ABB RobotStudio station: Task2_DONE_and_DEMOed.rspag

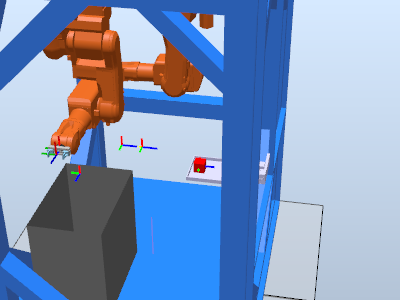
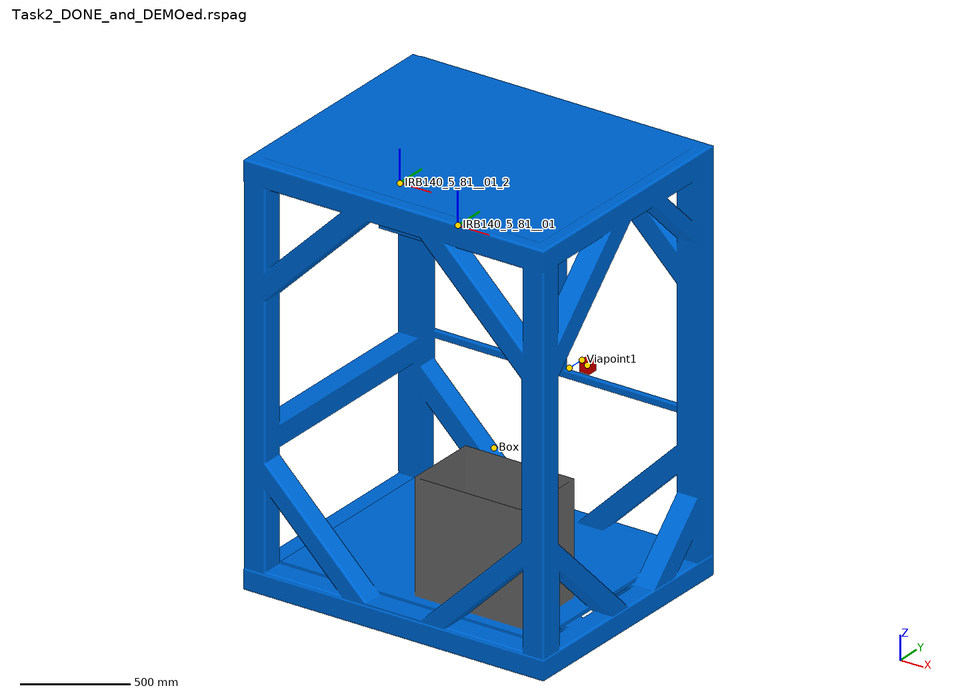
[picture v1: parts stored in the station drawn from their meshes, with robot base, taught points and paths (robot models come from the ABB library and are not in the file)]
--- station ---
Station LCFA_profile (saved by RobotStudio 22.2.10013.1)
Controller ALab_CellC_v1.0_4, task T_ROB2: task frame (RAPID world) sits at (78, -270, 2017) mm, rotated rx 180 ry 0 rz 0 deg in the station
Controller ALab_CellC_v1.0_4, task T_ROB1: task frame (RAPID world) sits at (78, -270, 2017) mm, rotated rx 180 ry 0 rz 0 deg in the station
Controller ALab_CellC_v1.0_4
  mechanical unit ROB_1: IRB140_5_81__01, 6 joints, base frame (0, 0, 0) mm
  mechanical unit ROB_2: IRB140_5_81__01_2, 6 joints, base frame (-596.17, -392.32, 108.97) mm, rotated rx -0.04 ry -0.66 rz 87.49 deg
Layout (positions relative to the parent item):
  - robotcage [part] at (0, 0, 87) mm, size 1670.4 x 1374.8 x 2180.4 mm
  - SampleTray [mechanism, from Libraries\SampleTray.rslib] at (263, 650, 160) mm; joint values [0] (rad or m)
  - IRB140_5_81__01 [mechanism, from Robots\IRB140_5_81__01.rslib] at (78, -270, 2017) mm, rotated rx 180 ry 0 rz 0 deg; joint values [0, 0, 0, 0, 0, 0] (rad or m)
  - IRB140_5_81__01_2 [mechanism, from Robots\IRB140_5_81__01.rslib] at (-518.17, 122.32, 1908.03) mm, rotated rx 179.96 ry 0.66 rz -87.49 deg; joint values [0, 0, 0, 0, 0, 0] (rad or m)
  - Gripper [mechanism, from Libraries\Gripper.rslib] at (593, -270, 1305) mm, rotated rx 0 ry -90 rz -180 deg; joint values [0] (rad or m)
  - Rubic Cube [part] at (76, 83.24, 1430.78) mm, rotated rx 180 ry 0 rz 90 deg, size 55 x 55 x 55 mm
  - Rubic Cube Simulation  [smart component]
      signals: DI DI_Open, DI DI_Close
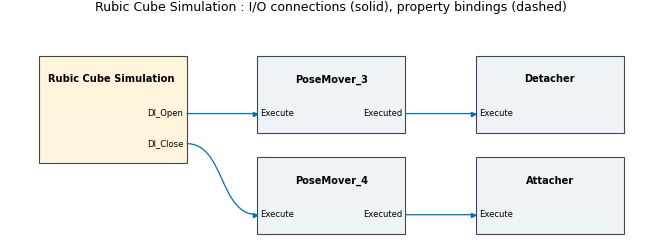
      connections:
        Rubic Cube Simulation .DI_Open -> PoseMover_3.Execute
        Rubic Cube Simulation .DI_Close -> PoseMover_4.Execute
        PoseMover_4.Executed -> Attacher.Execute
        PoseMover_3.Executed -> Detacher.Execute
    - PoseMover_3 [smart component, from Components\PoseMover.rslib]
        properties: Mechanism=Gripper; Pose=1; Duration=1
    - PoseMover_4 [smart component, from Components\PoseMover.rslib]
        properties: Mechanism=Gripper; Pose=2; Duration=1
    - Attacher [smart component, from Components\Attacher.rslib]
        properties: Parent=Gripper; Flange=0; Child=Rubic Cube; Mount=false; Offset=[0 0 0]; Orientation=[0 0 0]
    - Detacher [smart component, from Components\Detacher.rslib]
        properties: Child=Rubic Cube; KeepPosition=false
  - Box_1 [part] at (0, -500, 220) mm, size 600 x 400 x 0 mm
  - Box_2 [part] at (0, -500, 220) mm, rotated rx 90 ry 0 rz 0 deg, size 600 x 600 x 400 mm
  - Box_3 [part] at (0, -500, 820) mm, rotated rx 0 ry 90 rz 0 deg, size 600 x 400 x 600 mm
Attachment: Gripper is attached to IRB140_5_81__01 / Link6
EventTableEntry 4073: Group=, Trigger=AND 4074, Actions=[pose1 4075], Comment=, ActivationMode=2, Cyclic=false
EventTableTriggerLogic 4074: layoutX=167, layoutY=76, Operand1=AND 4076, Operand2=AND 4081, Operator=0, Delay=1000
EventTableActionIO 4075: IOValue=[-1], IRC5Controller=? -1, SignalTarget=LCFA_profile 1
EventTableTriggerLogic 4076: layoutX=94, layoutY=38, Operand1=cellC_gripper_horizontal_move 7096, Operand2=cellC_gripper_vertical_move 7097, Operator=0, Delay=1000
EventTableTriggerLogic 4081: layoutX=94, layoutY=109, Operand1=NOT 4082, Operand2=NOT 4084, Operator=0, Delay=1000
EventTableTriggerLogic 4082: layoutX=14, layoutY=96, Operand1=cellC_slider_horizontal_move 6338, Operand2=? -1, Operator=2, Delay=1000
EventTableTriggerLogic 4084: layoutX=9, layoutY=134, Operand1=cellC_slider_vertical_move 6339, Operand2=? -1, Operator=2, Delay=1000
EventTableEntry 4086: Group=, Trigger=AND 4087, Actions=[pose4 4097], Comment=, ActivationMode=2, Cyclic=false
EventTableTriggerLogic 4087: layoutX=194, layoutY=70, Operand1=AND 4088, Operand2=AND 4093, Operator=0, Delay=1000
EventTableTriggerLogic 4088: layoutX=73, layoutY=39, Operand1=cellC_gripper_horizontal_move 7098, Operand2=cellC_gripper_vertical_move 7099, Operator=0, Delay=1000
EventTableTriggerLogic 4093: layoutX=125, layoutY=101, Operand1=NOT 4094, Operand2=cellC_slider_vertical_move 6343, Operator=0, Delay=1000
EventTableTriggerLogic 4094: layoutX=19, layoutY=95, Operand1=cellC_slider_horizontal_move 6342, Operand2=? -1, Operator=2, Delay=1000
EventTableActionIO 4097: IOValue=[-1], IRC5Controller=? -1, SignalTarget=LCFA_profile 1
EventTableEntry 4098: Group=, Trigger=AND 4099, Actions=[pose8 4109], Comment=, ActivationMode=2, Cyclic=false
EventTableTriggerLogic 4099: layoutX=181, layoutY=88, Operand1=AND 4100, Operand2=AND 4105, Operator=0, Delay=1000
EventTableTriggerLogic 4100: layoutX=94, layoutY=47, Operand1=cellC_gripper_horizontal_move 7100, Operand2=cellC_gripper_vertical_move 7101, Operator=0, Delay=1000
EventTableTriggerLogic 4105: layoutX=92, layoutY=128, Operand1=cellC_slider_horizontal_move 6347, Operand2=NOT 4107, Operator=0, Delay=1000
EventTableTriggerLogic 4107: layoutX=18, layoutY=134, Operand1=cellC_slider_vertical_move 6346, Operand2=? -1, Operator=2, Delay=1000
EventTableActionIO 4109: IOValue=[-1], IRC5Controller=? -1, SignalTarget=LCFA_profile 1
EventTableEntry 4110: Group=, Trigger=AND 4111, Actions=[pose11 4120], Comment=, ActivationMode=2, Cyclic=false
EventTableTriggerLogic 4111: layoutX=165, layoutY=70, Operand1=AND 4112, Operand2=AND 4117, Operator=0, Delay=1000
EventTableTriggerLogic 4112: layoutX=93, layoutY=33, Operand1=cellC_gripper_horizontal_move 7102, Operand2=cellC_gripper_vertical_move 7103, Operator=0, Delay=1000
EventTableTriggerLogic 4117: layoutX=93, layoutY=131, Operand1=cellC_slider_horizontal_move 6350, Operand2=cellC_slider_vertical_move 6351, Operator=0, Delay=1000
EventTableActionIO 4120: IOValue=[-1], IRC5Controller=? -1, SignalTarget=LCFA_profile 1
EventTableEntry 4121: Group=, Trigger=AND 4122, Actions=[pose17 4132], Comment=, ActivationMode=2, Cyclic=false
EventTableTriggerLogic 4122: layoutX=217, layoutY=77, Operand1=AND 4123, Operand2=AND 4127, Operator=0, Delay=1000
EventTableTriggerLogic 4123: layoutX=119, layoutY=36, Operand1=cellC_gripper_horizontal_move 7960, Operand2=NOT 7105, Operator=0, Delay=1000
EventTableTriggerLogic 4127: layoutX=112, layoutY=96, Operand1=NOT 4128, Operand2=NOT 4130, Operator=0, Delay=1000
EventTableTriggerLogic 4128: layoutX=40, layoutY=96, Operand1=cellC_slider_horizontal_move 7961, Operand2=? -1, Operator=2, Delay=1000
EventTableTriggerLogic 4130: layoutX=35, layoutY=134, Operand1=cellC_slider_vertical_move 7962, Operand2=? -1, Operator=2, Delay=1000
EventTableActionIO 4132: IOValue=[-1], IRC5Controller=? -1, SignalTarget=LCFA_profile 1
EventTableEntry 4133: Group=, Trigger=AND 4134, Actions=[pose16 4143], Comment=, ActivationMode=2, Cyclic=false
EventTableTriggerLogic 4134: layoutX=168, layoutY=84, Operand1=AND 4135, Operand2=AND 4139, Operator=0, Delay=1000
EventTableTriggerLogic 4135: layoutX=90, layoutY=31, Operand1=cellC_gripper_horizontal_move 7106, Operand2=NOT 7107, Operator=0, Delay=1000
EventTableTriggerLogic 4139: layoutX=77, layoutY=109, Operand1=NOT 4253, Operand2=cellC_slider_vertical_move 6671, Operator=0, Delay=1000
EventTableActionIO 4143: IOValue=[-1], IRC5Controller=? -1, SignalTarget=LCFA_profile 1
EventTableEntry 4144: Group=, Trigger=AND 4145, Actions=[pose10 4154], Comment=, ActivationMode=2, Cyclic=false
EventTableTriggerLogic 4145: layoutX=219, layoutY=73, Operand1=AND 4146, Operand2=AND 4150, Operator=0, Delay=1000
EventTableTriggerLogic 4146: layoutX=143, layoutY=36, Operand1=cellC_gripper_horizontal_move 7964, Operand2=NOT 7110, Operator=0, Delay=1000
EventTableTriggerLogic 4150: layoutX=143, layoutY=107, Operand1=cellC_slider_horizontal_move 7966, Operand2=NOT 4152, Operator=0, Delay=1000
EventTableTriggerLogic 4152: layoutX=16, layoutY=136, Operand1=cellC_slider_vertical_move 7965, Operand2=? -1, Operator=2, Delay=1000
EventTableActionIO 4154: IOValue=[-1], IRC5Controller=? -1, SignalTarget=LCFA_profile 1
EventTableEntry 4155: Group=, Trigger=AND 4156, Actions=[pose14 4164], Comment=, ActivationMode=2, Cyclic=false
EventTableTriggerLogic 4156: layoutX=203, layoutY=67, Operand1=AND 4157, Operand2=AND 4161, Operator=0, Delay=1000
EventTableTriggerLogic 4157: layoutX=135, layoutY=41, Operand1=cellC_gripper_horizontal_move 7968, Operand2=NOT 7112, Operator=0, Delay=1000
EventTableTriggerLogic 4161: layoutX=132, layoutY=113, Operand1=cellC_slider_horizontal_move 7969, Operand2=cellC_slider_vertical_move 7970, Operator=0, Delay=1000
EventTableActionIO 4164: IOValue=[-1], IRC5Controller=? -1, SignalTarget=LCFA_profile 1
EventTableEntry 4165: Group=, Trigger=AND 4166, Actions=[pose2 4176], Comment=, ActivationMode=2, Cyclic=false
EventTableTriggerLogic 4166: layoutX=220, layoutY=69, Operand1=AND 4167, Operand2=AND 4171, Operator=0, Delay=1000
EventTableTriggerLogic 4167: layoutX=125, layoutY=14, Operand1=NOT 8003, Operand2=cellC_gripper_vertical_move 7972, Operator=0, Delay=1000
EventTableTriggerLogic 4171: layoutX=124, layoutY=95, Operand1=NOT 4172, Operand2=NOT 4174, Operator=0, Delay=1000
EventTableTriggerLogic 4172: layoutX=13, layoutY=97, Operand1=cellC_slider_horizontal_move 7973, Operand2=? -1, Operator=2, Delay=1000
EventTableTriggerLogic 4174: layoutX=11, layoutY=134, Operand1=cellC_slider_vertical_move 7974, Operand2=? -1, Operator=2, Delay=1000
EventTableActionIO 4176: IOValue=[-1], IRC5Controller=? -1, SignalTarget=LCFA_profile 1
EventTableEntry 4177: Group=, Trigger=AND 4178, Actions=[pose5 4187], Comment=, ActivationMode=2, Cyclic=false
EventTableTriggerLogic 4178: layoutX=243, layoutY=55, Operand1=AND 4179, Operand2=AND 4183, Operator=0, Delay=1000
EventTableTriggerLogic 4179: layoutX=162, layoutY=28, Operand1=NOT 8005, Operand2=cellC_gripper_vertical_move 7976, Operator=0, Delay=1000
EventTableTriggerLogic 4183: layoutX=173, layoutY=138, Operand1=NOT 4184, Operand2=cellC_slider_vertical_move 7978, Operator=0, Delay=1000
EventTableTriggerLogic 4184: layoutX=18, layoutY=95, Operand1=cellC_slider_horizontal_move 7977, Operand2=? -1, Operator=2, Delay=1000
EventTableActionIO 4187: IOValue=[-1], IRC5Controller=? -1, SignalTarget=LCFA_profile 1
EventTableEntry 4188: Group=, Trigger=AND 4189, Actions=[pose9 4198], Comment=, ActivationMode=2, Cyclic=false
EventTableTriggerLogic 4189: layoutX=204, layoutY=112, Operand1=AND 4190, Operand2=AND 4194, Operator=0, Delay=1000
EventTableTriggerLogic 4190: layoutX=108, layoutY=30, Operand1=NOT 8007, Operand2=cellC_gripper_vertical_move 7980, Operator=0, Delay=1000
EventTableTriggerLogic 4194: layoutX=108, layoutY=141, Operand1=cellC_slider_horizontal_move 7982, Operand2=NOT 4196, Operator=0, Delay=1000
EventTableTriggerLogic 4196: layoutX=26, layoutY=161, Operand1=cellC_slider_vertical_move 7981, Operand2=? -1, Operator=2, Delay=1000
EventTableActionIO 4198: IOValue=[-1], IRC5Controller=? -1, SignalTarget=LCFA_profile 1
EventTableEntry 4199: Group=, Trigger=AND 4200, Actions=[pose12 4208], Comment=, ActivationMode=2, Cyclic=false
EventTableTriggerLogic 4200: layoutX=245, layoutY=97, Operand1=AND 4201, Operand2=AND 4205, Operator=0, Delay=1000
EventTableTriggerLogic 4201: layoutX=182, layoutY=72, Operand1=NOT 8009, Operand2=cellC_gripper_vertical_move 7984, Operator=0, Delay=1000
EventTableTriggerLogic 4205: layoutX=189, layoutY=131, Operand1=cellC_slider_horizontal_move 7985, Operand2=cellC_slider_vertical_move 7986, Operator=0, Delay=1000
EventTableActionIO 4208: IOValue=[-1], IRC5Controller=? -1, SignalTarget=LCFA_profile 1
EventTableEntry 4209: Group=, Trigger=AND 4210, Actions=[pose3 4219], Comment=, ActivationMode=2, Cyclic=false
EventTableTriggerLogic 4210: layoutX=234, layoutY=61, Operand1=AND 4211, Operand2=AND 4214, Operator=0, Delay=1000
EventTableTriggerLogic 4211: layoutX=80, layoutY=23, Operand1=NOT 7117, Operand2=NOT 7118, Operator=0, Delay=1000
EventTableTriggerLogic 4214: layoutX=88, layoutY=113, Operand1=NOT 4215, Operand2=NOT 4217, Operator=0, Delay=1000
EventTableTriggerLogic 4215: layoutX=16, layoutY=85, Operand1=cellC_slider_horizontal_move 7989, Operand2=? -1, Operator=2, Delay=1000
EventTableTriggerLogic 4217: layoutX=33, layoutY=125, Operand1=cellC_slider_vertical_move 7990, Operand2=? -1, Operator=2, Delay=1000
EventTableActionIO 4219: IOValue=[-1], IRC5Controller=? -1, SignalTarget=LCFA_profile 1
EventTableEntry 4220: Group=, Trigger=AND 4221, Actions=[pose6 4229], Comment=, ActivationMode=2, Cyclic=false
EventTableTriggerLogic 4221: layoutX=192, layoutY=87, Operand1=AND 4222, Operand2=AND 4225, Operator=0, Delay=1000
EventTableTriggerLogic 4222: layoutX=118, layoutY=38, Operand1=NOT 7119, Operand2=NOT 7120, Operator=0, Delay=1000
EventTableTriggerLogic 4225: layoutX=113, layoutY=118, Operand1=NOT 4226, Operand2=cellC_slider_vertical_move 7994, Operator=0, Delay=1000
EventTableTriggerLogic 4226: layoutX=14, layoutY=101, Operand1=cellC_slider_horizontal_move 7993, Operand2=? -1, Operator=2, Delay=1000
EventTableActionIO 4229: IOValue=[-1], IRC5Controller=? -1, SignalTarget=LCFA_profile 1
EventTableEntry 4230: Group=, Trigger=AND 4231, Actions=[pose7 4239], Comment=, ActivationMode=2, Cyclic=false
EventTableTriggerLogic 4231: layoutX=212, layoutY=64, Operand1=AND 4232, Operand2=AND 4235, Operator=0, Delay=1000
EventTableTriggerLogic 4232: layoutX=113, layoutY=37, Operand1=NOT 7121, Operand2=NOT 7122, Operator=0, Delay=1000
EventTableTriggerLogic 4235: layoutX=113, layoutY=104, Operand1=cellC_slider_horizontal_move 7998, Operand2=NOT 4237, Operator=0, Delay=1000
EventTableTriggerLogic 4237: layoutX=13, layoutY=128, Operand1=cellC_slider_vertical_move 7997, Operand2=? -1, Operator=2, Delay=1000
EventTableActionIO 4239: IOValue=[-1], IRC5Controller=? -1, SignalTarget=LCFA_profile 1
EventTableEntry 4240: Group=, Trigger=AND 4241, Actions=[pose13 4248], Comment=, ActivationMode=2, Cyclic=false
EventTableTriggerLogic 4241: layoutX=160, layoutY=73, Operand1=AND 4242, Operand2=AND 4245, Operator=0, Delay=1000
EventTableTriggerLogic 4242: layoutX=68, layoutY=38, Operand1=NOT 7123, Operand2=NOT 7124, Operator=0, Delay=1000
EventTableTriggerLogic 4245: layoutX=67, layoutY=107, Operand1=cellC_slider_horizontal_move 8001, Operand2=cellC_slider_vertical_move 8002, Operator=0, Delay=1000
EventTableActionIO 4248: IOValue=[-1], IRC5Controller=? -1, SignalTarget=LCFA_profile 1
EventTableTriggerLogic 4253: layoutX=22, layoutY=89, Operand1=cellC_slider_horizontal_move 6670, Operand2=? -1, Operator=2, Delay=1000
EventTableEntry 4262: Group=, Trigger=AND 4263, Actions=[conv1_buffer6 4271], Comment=, ActivationMode=2, Cyclic=false
EventTableTriggerLogic 4263: layoutX=153, layoutY=73, Operand1=AND 4264, Operand2=NOT 4269, Operator=0, Delay=1000
EventTableTriggerLogic 4264: layoutX=80, layoutY=34, Operand1=NOT 4265, Operand2=NOT 4267, Operator=0, Delay=1000
EventTableTriggerLogic 4265: layoutX=8, layoutY=16, Operand1=conv1_buffer_horizontal_open 6327, Operand2=? -1, Operator=2, Delay=1000
EventTableTriggerLogic 4267: layoutX=9, layoutY=52, Operand1=conv1_buffer_lower_go_up 6328, Operand2=? -1, Operator=2, Delay=1000
EventTableTriggerLogic 4269: layoutX=9, layoutY=86, Operand1=conv1_buffer_upper_go_down 6329, Operand2=? -1, Operator=2, Delay=1000
EventTableActionIO 4271: IOValue=[-1], IRC5Controller=? -1, SignalTarget=LCFA_profile 1
EventTableEntry 4272: Group=, Trigger=AND 4273, Actions=[conv1_buffer5 4280], Comment=, ActivationMode=2, Cyclic=false
EventTableTriggerLogic 4273: layoutX=133, layoutY=81, Operand1=AND 4274, Operand2=conv1_buffer_upper_go_down 6332, Operator=0, Delay=1000
EventTableTriggerLogic 4274: layoutX=93, layoutY=26, Operand1=NOT 4275, Operand2=NOT 4277, Operator=0, Delay=1000
EventTableTriggerLogic 4275: layoutX=8, layoutY=16, Operand1=conv1_buffer_horizontal_open 6330, Operand2=? -1, Operator=2, Delay=1000
EventTableTriggerLogic 4277: layoutX=9, layoutY=53, Operand1=conv1_buffer_lower_go_up 6331, Operand2=? -1, Operator=2, Delay=1000
EventTableActionIO 4280: IOValue=[-1], IRC5Controller=? -1, SignalTarget=LCFA_profile 1
EventTableEntry 4281: Group=, Trigger=AND 4282, Actions=[conv1_buffer8 4289], Comment=, ActivationMode=2, Cyclic=false
EventTableTriggerLogic 4282: layoutX=184, layoutY=91, Operand1=AND 4283, Operand2=NOT 4287, Operator=0, Delay=1000
EventTableTriggerLogic 4283: layoutX=106, layoutY=52, Operand1=NOT 4284, Operand2=conv1_buffer_lower_go_up 6334, Operator=0, Delay=1000
EventTableTriggerLogic 4284: layoutX=13, layoutY=17, Operand1=conv1_buffer_horizontal_open 6333, Operand2=? -1, Operator=2, Delay=1000
EventTableTriggerLogic 4287: layoutX=23, layoutY=94, Operand1=conv1_buffer_upper_go_down 6335, Operand2=? -1, Operator=2, Delay=1000
EventTableActionIO 4289: IOValue=[-1], IRC5Controller=? -1, SignalTarget=LCFA_profile 1
EventTableEntry 4290: Group=, Trigger=AND 4291, Actions=[conv1_buffer7 4297], Comment=, ActivationMode=2, Cyclic=false
EventTableTriggerLogic 4291: layoutX=211, layoutY=90, Operand1=AND 4292, Operand2=conv1_buffer_upper_go_down 6282, Operator=0, Delay=1000
EventTableTriggerLogic 4292: layoutX=106, layoutY=24, Operand1=NOT 4293, Operand2=conv1_buffer_lower_go_up 6281, Operator=0, Delay=1000
EventTableTriggerLogic 4293: layoutX=35, layoutY=17, Operand1=conv1_buffer_horizontal_open 6280, Operand2=? -1, Operator=2, Delay=1000
EventTableActionIO 4297: IOValue=[-1], IRC5Controller=? -1, SignalTarget=LCFA_profile 1
EventTableEntry 4298: Group=, Trigger=AND 4299, Actions=[conv1_buffer2 4306], Comment=, ActivationMode=2, Cyclic=false
EventTableTriggerLogic 4299: layoutX=226, layoutY=110, Operand1=AND 4300, Operand2=NOT 4304, Operator=0, Delay=1000
EventTableTriggerLogic 4300: layoutX=93, layoutY=30, Operand1=conv1_buffer_horizontal_open 6284, Operand2=NOT 4302, Operator=0, Delay=1000
EventTableTriggerLogic 4302: layoutX=30, layoutY=56, Operand1=conv1_buffer_lower_go_up 6283, Operand2=? -1, Operator=2, Delay=1000
EventTableTriggerLogic 4304: layoutX=17, layoutY=96, Operand1=conv1_buffer_upper_go_down 6285, Operand2=? -1, Operator=2, Delay=1000
EventTableActionIO 4306: IOValue=[-1], IRC5Controller=? -1, SignalTarget=LCFA_profile 1
EventTableEntry 4307: Group=, Trigger=AND 4308, Actions=[conv1_buffer1 4314], Comment=, ActivationMode=2, Cyclic=false
EventTableTriggerLogic 4308: layoutX=164, layoutY=68, Operand1=AND 4309, Operand2=conv1_buffer_upper_go_down 6288, Operator=0, Delay=1000
EventTableTriggerLogic 4309: layoutX=96, layoutY=16, Operand1=conv1_buffer_horizontal_open 6287, Operand2=NOT 4311, Operator=0, Delay=1000
EventTableTriggerLogic 4311: layoutX=18, layoutY=46, Operand1=conv1_buffer_lower_go_up 6286, Operand2=? -1, Operator=2, Delay=1000
EventTableActionIO 4314: IOValue=[-1], IRC5Controller=? -1, SignalTarget=LCFA_profile 1
EventTableEntry 4315: Group=, Trigger=AND 4316, Actions=[conv1_buffer4 4322], Comment=, ActivationMode=2, Cyclic=false
EventTableTriggerLogic 4316: layoutX=161, layoutY=63, Operand1=AND 4317, Operand2=NOT 4320, Operator=0, Delay=1000
EventTableTriggerLogic 4317: layoutX=52, layoutY=16, Operand1=conv1_buffer_horizontal_open 6289, Operand2=conv1_buffer_lower_go_up 6290, Operator=0, Delay=1000
EventTableTriggerLogic 4320: layoutX=26, layoutY=137, Operand1=conv1_buffer_upper_go_down 6291, Operand2=? -1, Operator=2, Delay=1000
EventTableActionIO 4322: IOValue=[-1], IRC5Controller=? -1, SignalTarget=LCFA_profile 1
EventTableEntry 4323: Group=, Trigger=AND 4324, Actions=[conv1_buffer3 4329], Comment=, ActivationMode=2, Cyclic=false
EventTableTriggerLogic 4324: layoutX=174, layoutY=87, Operand1=AND 4325, Operand2=conv1_buffer_upper_go_down 6294, Operator=0, Delay=1000
EventTableTriggerLogic 4325: layoutX=74, layoutY=31, Operand1=conv1_buffer_horizontal_open 6292, Operand2=conv1_buffer_lower_go_up 6293, Operator=0, Delay=1000
EventTableActionIO 4329: IOValue=[-1], IRC5Controller=? -1, SignalTarget=LCFA_profile 1
EventTableEntry 4330: Group=, Trigger=AND 4331, Actions=[conv2_buffer6 4339], Comment=, ActivationMode=2, Cyclic=false
EventTableTriggerLogic 4331: layoutX=148, layoutY=98, Operand1=AND 4332, Operand2=NOT 4337, Operator=0, Delay=1000
EventTableTriggerLogic 4332: layoutX=101, layoutY=54, Operand1=NOT 4333, Operand2=NOT 4335, Operator=0, Delay=1000
EventTableTriggerLogic 4333: layoutX=31, layoutY=17, Operand1=conv2_buffer_horizontal_move 6295, Operand2=? -1, Operator=2, Delay=1000
EventTableTriggerLogic 4335: layoutX=32, layoutY=53, Operand1=conv2_buffer_lower_vertical_move 6296, Operand2=? -1, Operator=2, Delay=1000
EventTableTriggerLogic 4337: layoutX=31, layoutY=89, Operand1=conv2_buffer_upper_vertical_move 6297, Operand2=? -1, Operator=2, Delay=1000
EventTableActionIO 4339: IOValue=[-1], IRC5Controller=? -1, SignalTarget=LCFA_profile 1
EventTableEntry 4340: Group=, Trigger=AND 4341, Actions=[conv2_buffer5 4348], Comment=, ActivationMode=2, Cyclic=false
EventTableTriggerLogic 4341: layoutX=206, layoutY=74, Operand1=AND 4342, Operand2=conv2_buffer_upper_vertical_move 6300, Operator=0, Delay=1000
EventTableTriggerLogic 4342: layoutX=94, layoutY=37, Operand1=NOT 4343, Operand2=NOT 4345, Operator=0, Delay=1000
EventTableTriggerLogic 4343: layoutX=13, layoutY=14, Operand1=conv2_buffer_horizontal_move 6298, Operand2=? -1, Operator=2, Delay=1000
EventTableTriggerLogic 4345: layoutX=9, layoutY=56, Operand1=conv2_buffer_lower_vertical_move 6299, Operand2=? -1, Operator=2, Delay=1000
EventTableActionIO 4348: IOValue=[-1], IRC5Controller=? -1, SignalTarget=LCFA_profile 1
EventTableEntry 4349: Group=, Trigger=AND 4350, Actions=[conv2_buffer8 4357], Comment=, ActivationMode=2, Cyclic=false
EventTableTriggerLogic 4350: layoutX=195, layoutY=82, Operand1=AND 4351, Operand2=NOT 4355, Operator=0, Delay=1000
EventTableTriggerLogic 4351: layoutX=67, layoutY=49, Operand1=NOT 4352, Operand2=conv2_buffer_lower_vertical_move 6302, Operator=0, Delay=1000
EventTableTriggerLogic 4352: layoutX=20, layoutY=15, Operand1=conv2_buffer_horizontal_move 6301, Operand2=? -1, Operator=2, Delay=1000
EventTableTriggerLogic 4355: layoutX=20, layoutY=92, Operand1=conv2_buffer_upper_vertical_move 6303, Operand2=? -1, Operator=2, Delay=1000
EventTableActionIO 4357: IOValue=[-1], IRC5Controller=? -1, SignalTarget=LCFA_profile 1
EventTableEntry 4358: Group=, Trigger=AND 4359, Actions=[conv2_buffer7 4365], Comment=, ActivationMode=2, Cyclic=false
EventTableTriggerLogic 4359: layoutX=193, layoutY=94, Operand1=AND 4360, Operand2=conv2_buffer_upper_vertical_move 6306, Operator=0, Delay=1000
EventTableTriggerLogic 4360: layoutX=111, layoutY=44, Operand1=NOT 4361, Operand2=conv2_buffer_lower_vertical_move 6305, Operator=0, Delay=1000
EventTableTriggerLogic 4361: layoutX=48, layoutY=16, Operand1=conv2_buffer_horizontal_move 6304, Operand2=? -1, Operator=2, Delay=1000
EventTableActionIO 4365: IOValue=[-1], IRC5Controller=? -1, SignalTarget=LCFA_profile 1
EventTableEntry 4366: Group=, Trigger=AND 4367, Actions=[conv2_buffer2 4374], Comment=, ActivationMode=2, Cyclic=false
EventTableTriggerLogic 4367: layoutX=210, layoutY=27, Operand1=conv2_buffer_horizontal_move 6309, Operand2=AND 4369, Operator=0, Delay=1000
EventTableTriggerLogic 4369: layoutX=163, layoutY=91, Operand1=NOT 4370, Operand2=NOT 4372, Operator=0, Delay=1000
EventTableTriggerLogic 4370: layoutX=21, layoutY=58, Operand1=conv2_buffer_lower_vertical_move 6307, Operand2=? -1, Operator=2, Delay=1000
EventTableTriggerLogic 4372: layoutX=24, layoutY=96, Operand1=conv2_buffer_upper_vertical_move 6308, Operand2=? -1, Operator=2, Delay=1000
EventTableActionIO 4374: IOValue=[-1], IRC5Controller=? -1, SignalTarget=LCFA_profile 1
EventTableEntry 4375: Group=, Trigger=AND 4376, Actions=[conv2_buffer1 4382], Comment=, ActivationMode=2, Cyclic=false
EventTableTriggerLogic 4376: layoutX=233, layoutY=95, Operand1=AND 4377, Operand2=conv2_buffer_upper_vertical_move 6312, Operator=0, Delay=1000
EventTableTriggerLogic 4377: layoutX=160, layoutY=50, Operand1=conv2_buffer_horizontal_move 6311, Operand2=NOT 4379, Operator=0, Delay=1000
EventTableTriggerLogic 4379: layoutX=37, layoutY=56, Operand1=conv2_buffer_lower_vertical_move 6310, Operand2=? -1, Operator=2, Delay=1000
EventTableActionIO 4382: IOValue=[-1], IRC5Controller=? -1, SignalTarget=LCFA_profile 1
EventTableEntry 4383: Group=, Trigger=AND 4384, Actions=[conv2_buffer4 4390], Comment=, ActivationMode=2, Cyclic=false
EventTableTriggerLogic 4384: layoutX=102, layoutY=69, Operand1=AND 4385, Operand2=NOT 4388, Operator=0, Delay=1000
EventTableTriggerLogic 4385: layoutX=32, layoutY=42, Operand1=conv2_buffer_horizontal_move 6313, Operand2=conv2_buffer_lower_vertical_move 6314, Operator=0, Delay=1000
EventTableTriggerLogic 4388: layoutX=24, layoutY=96, Operand1=conv2_buffer_upper_vertical_move 6315, Operand2=? -1, Operator=2, Delay=1000
EventTableActionIO 4390: IOValue=[-1], IRC5Controller=? -1, SignalTarget=LCFA_profile 1
EventTableEntry 4391: Group=, Trigger=AND 4392, Actions=[conv2_buffer3 4397], Comment=, ActivationMode=2, Cyclic=false
EventTableTriggerLogic 4392: layoutX=97, layoutY=92, Operand1=AND 4393, Operand2=conv2_buffer_upper_vertical_move 6318, Operator=0, Delay=1000
EventTableTriggerLogic 4393: layoutX=42, layoutY=52, Operand1=conv2_buffer_horizontal_move 6316, Operand2=conv2_buffer_lower_vertical_move 6317, Operator=0, Delay=1000
EventTableActionIO 4397: IOValue=[-1], IRC5Controller=? -1, SignalTarget=LCFA_profile 1
EventTableEntry 4398: Group=, Trigger=AND 4399, Actions=[palletHolder1 4404], Comment=, ActivationMode=2, Cyclic=false
EventTableTriggerLogic 4399: layoutX=96, layoutY=16, Operand1=cellC_pallet_holder 7125, Operand2=cellC_pallet_stopper 7126, Operator=0, Delay=1000
EventTableActionIO 4404: IOValue=[-1], IRC5Controller=? -1, SignalTarget=LCFA_profile 1
EventTableEntry 4405: Group=, Trigger=AND 4406, Actions=[palletHolder2 4410], Comment=, ActivationMode=2, Cyclic=false
EventTableTriggerLogic 4406: layoutX=142, layoutY=32, Operand1=NOT 7128, Operand2=cellC_pallet_stopper 7127, Operator=0, Delay=1000
EventTableActionIO 4410: IOValue=[-1], IRC5Controller=? -1, SignalTarget=LCFA_profile 1
EventTableEntry 4411: Group=, Trigger=AND 4412, Actions=[palletHolder4 4415], Comment=, ActivationMode=2, Cyclic=false
EventTableTriggerLogic 4412: layoutX=51, layoutY=46, Operand1=NOT 7130, Operand2=NOT 7132, Operator=0, Delay=1000
EventTableActionIO 4415: IOValue=[-1], IRC5Controller=? -1, SignalTarget=LCFA_profile 1
EventTableEntry 4416: Group=, Trigger=AND 4417, Actions=[palletHolder3 4419], Comment=, ActivationMode=2, Cyclic=false
EventTableTriggerLogic 4417: layoutX=107, layoutY=60, Operand1=cellC_pallet_holder 7134, Operand2=NOT 7135, Operator=0, Delay=1000
EventTableActionIO 4419: IOValue=[-1], IRC5Controller=? -1, SignalTarget=LCFA_profile 1
EventTableEntry 4425: Group=, Trigger=TestPlateDrive 4426, Actions=[EventTableActionMechanicalPose 4427], Comment=, ActivationMode=2, Cyclic=false
EventTableTriggerIO 4426: IOValue=[1], IRC5Controller=? -1, Operator=0, SignalSource=ALab_CellC_v1.0_4 5362
EventTableActionMechanicalPose 4427: VirtualSignal=, Mechanism=SampleTray 568, ToPoseName=HomePosition, VirtualSignalValue=[1]
EventTableTriggerIO 6280: IOValue=[-1], IRC5Controller=? -1, Operator=0, SignalSource=ALab_CellC_v1.0_4 5362
EventTableTriggerIO 6281: IOValue=[-1], IRC5Controller=? -1, Operator=0, SignalSource=ALab_CellC_v1.0_4 5362
EventTableTriggerIO 6282: IOValue=[-1], IRC5Controller=? -1, Operator=0, SignalSource=ALab_CellC_v1.0_4 5362
EventTableTriggerIO 6283: IOValue=[-1], IRC5Controller=? -1, Operator=0, SignalSource=ALab_CellC_v1.0_4 5362
EventTableTriggerIO 6284: IOValue=[-1], IRC5Controller=? -1, Operator=0, SignalSource=ALab_CellC_v1.0_4 5362
EventTableTriggerIO 6285: IOValue=[-1], IRC5Controller=? -1, Operator=0, SignalSource=ALab_CellC_v1.0_4 5362
EventTableTriggerIO 6286: IOValue=[-1], IRC5Controller=? -1, Operator=0, SignalSource=ALab_CellC_v1.0_4 5362
EventTableTriggerIO 6287: IOValue=[-1], IRC5Controller=? -1, Operator=0, SignalSource=ALab_CellC_v1.0_4 5362
EventTableTriggerIO 6288: IOValue=[-1], IRC5Controller=? -1, Operator=0, SignalSource=ALab_CellC_v1.0_4 5362
EventTableTriggerIO 6289: IOValue=[-1], IRC5Controller=? -1, Operator=0, SignalSource=ALab_CellC_v1.0_4 5362
EventTableTriggerIO 6290: IOValue=[-1], IRC5Controller=? -1, Operator=0, SignalSource=ALab_CellC_v1.0_4 5362
EventTableTriggerIO 6291: IOValue=[-1], IRC5Controller=? -1, Operator=0, SignalSource=ALab_CellC_v1.0_4 5362
EventTableTriggerIO 6292: IOValue=[-1], IRC5Controller=? -1, Operator=0, SignalSource=ALab_CellC_v1.0_4 5362
EventTableTriggerIO 6293: IOValue=[-1], IRC5Controller=? -1, Operator=0, SignalSource=ALab_CellC_v1.0_4 5362
EventTableTriggerIO 6294: IOValue=[-1], IRC5Controller=? -1, Operator=0, SignalSource=ALab_CellC_v1.0_4 5362
EventTableTriggerIO 6295: IOValue=[-1], IRC5Controller=? -1, Operator=0, SignalSource=ALab_CellC_v1.0_4 5362
EventTableTriggerIO 6296: IOValue=[-1], IRC5Controller=? -1, Operator=0, SignalSource=ALab_CellC_v1.0_4 5362
EventTableTriggerIO 6297: IOValue=[-1], IRC5Controller=? -1, Operator=0, SignalSource=ALab_CellC_v1.0_4 5362
EventTableTriggerIO 6298: IOValue=[-1], IRC5Controller=? -1, Operator=0, SignalSource=ALab_CellC_v1.0_4 5362
EventTableTriggerIO 6299: IOValue=[-1], IRC5Controller=? -1, Operator=0, SignalSource=ALab_CellC_v1.0_4 5362
EventTableTriggerIO 6300: IOValue=[-1], IRC5Controller=? -1, Operator=0, SignalSource=ALab_CellC_v1.0_4 5362
EventTableTriggerIO 6301: IOValue=[-1], IRC5Controller=? -1, Operator=0, SignalSource=ALab_CellC_v1.0_4 5362
EventTableTriggerIO 6302: IOValue=[-1], IRC5Controller=? -1, Operator=0, SignalSource=ALab_CellC_v1.0_4 5362
EventTableTriggerIO 6303: IOValue=[-1], IRC5Controller=? -1, Operator=0, SignalSource=ALab_CellC_v1.0_4 5362
EventTableTriggerIO 6304: IOValue=[-1], IRC5Controller=? -1, Operator=0, SignalSource=ALab_CellC_v1.0_4 5362
EventTableTriggerIO 6305: IOValue=[-1], IRC5Controller=? -1, Operator=0, SignalSource=ALab_CellC_v1.0_4 5362
EventTableTriggerIO 6306: IOValue=[-1], IRC5Controller=? -1, Operator=0, SignalSource=ALab_CellC_v1.0_4 5362
EventTableTriggerIO 6307: IOValue=[-1], IRC5Controller=? -1, Operator=0, SignalSource=ALab_CellC_v1.0_4 5362
EventTableTriggerIO 6308: IOValue=[-1], IRC5Controller=? -1, Operator=0, SignalSource=ALab_CellC_v1.0_4 5362
EventTableTriggerIO 6309: IOValue=[-1], IRC5Controller=? -1, Operator=0, SignalSource=ALab_CellC_v1.0_4 5362
EventTableTriggerIO 6310: IOValue=[-1], IRC5Controller=? -1, Operator=0, SignalSource=ALab_CellC_v1.0_4 5362
EventTableTriggerIO 6311: IOValue=[-1], IRC5Controller=? -1, Operator=0, SignalSource=ALab_CellC_v1.0_4 5362
EventTableTriggerIO 6312: IOValue=[-1], IRC5Controller=? -1, Operator=0, SignalSource=ALab_CellC_v1.0_4 5362
EventTableTriggerIO 6313: IOValue=[-1], IRC5Controller=? -1, Operator=0, SignalSource=ALab_CellC_v1.0_4 5362
EventTableTriggerIO 6314: IOValue=[-1], IRC5Controller=? -1, Operator=0, SignalSource=ALab_CellC_v1.0_4 5362
EventTableTriggerIO 6315: IOValue=[-1], IRC5Controller=? -1, Operator=0, SignalSource=ALab_CellC_v1.0_4 5362
EventTableTriggerIO 6316: IOValue=[-1], IRC5Controller=? -1, Operator=0, SignalSource=ALab_CellC_v1.0_4 5362
EventTableTriggerIO 6317: IOValue=[-1], IRC5Controller=? -1, Operator=0, SignalSource=ALab_CellC_v1.0_4 5362
EventTableTriggerIO 6318: IOValue=[-1], IRC5Controller=? -1, Operator=0, SignalSource=ALab_CellC_v1.0_4 5362
EventTableTriggerIO 6327: IOValue=[-1], IRC5Controller=? -1, Operator=0, SignalSource=ALab_CellC_v1.0_4 5362
EventTableTriggerIO 6328: IOValue=[-1], IRC5Controller=? -1, Operator=0, SignalSource=ALab_CellC_v1.0_4 5362
EventTableTriggerIO 6329: IOValue=[-1], IRC5Controller=? -1, Operator=0, SignalSource=ALab_CellC_v1.0_4 5362
EventTableTriggerIO 6330: IOValue=[-1], IRC5Controller=? -1, Operator=0, SignalSource=ALab_CellC_v1.0_4 5362
EventTableTriggerIO 6331: IOValue=[-1], IRC5Controller=? -1, Operator=0, SignalSource=ALab_CellC_v1.0_4 5362
EventTableTriggerIO 6332: IOValue=[-1], IRC5Controller=? -1, Operator=0, SignalSource=ALab_CellC_v1.0_4 5362
EventTableTriggerIO 6333: IOValue=[-1], IRC5Controller=? -1, Operator=0, SignalSource=ALab_CellC_v1.0_4 5362
EventTableTriggerIO 6334: IOValue=[-1], IRC5Controller=? -1, Operator=0, SignalSource=ALab_CellC_v1.0_4 5362
EventTableTriggerIO 6335: IOValue=[-1], IRC5Controller=? -1, Operator=0, SignalSource=ALab_CellC_v1.0_4 5362
EventTableTriggerIO 6338: IOValue=[-1], IRC5Controller=? -1, Operator=0, SignalSource=ALab_CellC_v1.0_4 5362
EventTableTriggerIO 6339: IOValue=[-1], IRC5Controller=? -1, Operator=0, SignalSource=ALab_CellC_v1.0_4 5362
EventTableTriggerIO 6342: IOValue=[-1], IRC5Controller=? -1, Operator=0, SignalSource=ALab_CellC_v1.0_4 5362
EventTableTriggerIO 6343: IOValue=[-1], IRC5Controller=? -1, Operator=0, SignalSource=ALab_CellC_v1.0_4 5362
EventTableTriggerIO 6346: IOValue=[-1], IRC5Controller=? -1, Operator=0, SignalSource=ALab_CellC_v1.0_4 5362
EventTableTriggerIO 6347: IOValue=[-1], IRC5Controller=? -1, Operator=0, SignalSource=ALab_CellC_v1.0_4 5362
EventTableTriggerIO 6350: IOValue=[-1], IRC5Controller=? -1, Operator=0, SignalSource=ALab_CellC_v1.0_4 5362
EventTableTriggerIO 6351: IOValue=[-1], IRC5Controller=? -1, Operator=0, SignalSource=ALab_CellC_v1.0_4 5362
EventTableEntry 6400: Group=, Trigger=AND 6401, Actions=[PalletIO00 6413], Comment=, ActivationMode=2, Cyclic=false
EventTableTriggerLogic 6401: layoutX=184, layoutY=128, Operand1=AND 6402, Operand2=AND 6408, Operator=0, Delay=1000
EventTableTriggerLogic 6402: layoutX=119, layoutY=95, Operand1=AND 6403, Operand2=conv1_outer_lifter 6407, Operator=0, Delay=1000
EventTableTriggerLogic 6403: layoutX=72, layoutY=30, Operand1=conv1_motor_s1 6404, Operand2=NOT 6405, Operator=0, Delay=1000
EventTableTriggerIO 6404: IOValue=[-1], IRC5Controller=? -1, Operator=0, SignalSource=ALab_CellC_v1.0_4 5362
EventTableTriggerLogic 6405: layoutX=22, layoutY=51, Operand1=conv1_motor_s2 6406, Operand2=? -1, Operator=2, Delay=1000
EventTableTriggerIO 6406: IOValue=[-1], IRC5Controller=? -1, Operator=0, SignalSource=ALab_CellC_v1.0_4 5362
EventTableTriggerIO 6407: IOValue=[-1], IRC5Controller=? -1, Operator=0, SignalSource=ALab_CellC_v1.0_4 5362
EventTableTriggerLogic 6408: layoutX=108, layoutY=144, Operand1=NOT 6409, Operand2=NOT 6411, Operator=0, Delay=1000
EventTableTriggerLogic 6409: layoutX=26, layoutY=126, Operand1=conv2_motor_s1 6410, Operand2=? -1, Operator=2, Delay=1000
EventTableTriggerIO 6410: IOValue=[-1], IRC5Controller=? -1, Operator=0, SignalSource=ALab_CellC_v1.0_4 5362
EventTableTriggerLogic 6411: layoutX=31, layoutY=161, Operand1=conv2_motor_s2 6412, Operand2=? -1, Operator=2, Delay=1000
EventTableTriggerIO 6412: IOValue=[-1], IRC5Controller=? -1, Operator=0, SignalSource=ALab_CellC_v1.0_4 5362
EventTableActionIO 6413: IOValue=[-1], IRC5Controller=? -1, SignalTarget=LCFA_profile 1
EventTableEntry 6414: Group=, Trigger=AND 6415, Actions=[PalletIO2 6427], Comment=, ActivationMode=2, Cyclic=false
EventTableTriggerLogic 6415: layoutX=231, layoutY=144, Operand1=AND 6416, Operand2=pallet1 6426, Operator=0, Delay=1000
EventTableTriggerLogic 6416: layoutX=170, layoutY=83, Operand1=AND 6417, Operand2=AND 6421, Operator=0, Delay=1000
EventTableTriggerLogic 6417: layoutX=104, layoutY=35, Operand1=conv1_motor_s1 6418, Operand2=NOT 6419, Operator=0, Delay=1000
EventTableTriggerIO 6418: IOValue=[-1], IRC5Controller=? -1, Operator=0, SignalSource=ALab_CellC_v1.0_4 5362
EventTableTriggerLogic 6419: layoutX=20, layoutY=57, Operand1=conv1_motor_s2 6420, Operand2=? -1, Operator=2, Delay=1000
EventTableTriggerIO 6420: IOValue=[-1], IRC5Controller=? -1, Operator=0, SignalSource=ALab_CellC_v1.0_4 5362
EventTableTriggerLogic 6421: layoutX=96, layoutY=120, Operand1=NOT 6422, Operand2=NOT 6424, Operator=0, Delay=1000
EventTableTriggerLogic 6422: layoutX=19, layoutY=94, Operand1=conv2_motor_s1 6423, Operand2=? -1, Operator=2, Delay=1000
EventTableTriggerIO 6423: IOValue=[-1], IRC5Controller=? -1, Operator=0, SignalSource=ALab_CellC_v1.0_4 5362
EventTableTriggerLogic 6424: layoutX=20, layoutY=128, Operand1=conv2_motor_s2 6425, Operand2=? -1, Operator=2, Delay=1000
EventTableTriggerIO 6425: IOValue=[-1], IRC5Controller=? -1, Operator=0, SignalSource=ALab_CellC_v1.0_4 5362
EventTableTriggerIO 6426: IOValue=[-1], IRC5Controller=? -1, Operator=0, SignalSource=LCFA_profile 1
EventTableActionIO 6427: IOValue=[-1], IRC5Controller=? -1, SignalTarget=LCFA_profile 1
EventTableEntry 6428: Group=, Trigger=AND 8113, Actions=[PalletIO4 6443], Comment=, ActivationMode=2, Cyclic=false
EventTableActionIO 6443: IOValue=[-1], IRC5Controller=? -1, SignalTarget=LCFA_profile 1
EventTableEntry 6444: Group=, Trigger=AND 6445, Actions=[PalletIO3 6448], Comment=, ActivationMode=2, Cyclic=false
EventTableTriggerLogic 6445: layoutX=62, layoutY=38, Operand1=pallet2 8126, Operand2=cellC_slider_horizontal_move 8125, Operator=0, Delay=1000
EventTableActionIO 6448: IOValue=[-1], IRC5Controller=? -1, SignalTarget=LCFA_profile 1
EventTableEntry 6449: Group=, Trigger=AND 6450, Actions=[PalletIO5 6453], Comment=, ActivationMode=2, Cyclic=false
EventTableTriggerLogic 6450: layoutX=133, layoutY=37, Operand1=pallet3 6451, Operand2=pose6 6452, Operator=0, Delay=1000
EventTableTriggerIO 6451: IOValue=[-1], IRC5Controller=? -1, Operator=0, SignalSource=LCFA_profile 1
EventTableTriggerIO 6452: IOValue=[-1], IRC5Controller=? -1, Operator=0, SignalSource=LCFA_profile 1
EventTableActionIO 6453: IOValue=[-1], IRC5Controller=? -1, SignalTarget=LCFA_profile 1
EventTableEntry 6454: Group=, Trigger=AND 6455, Actions=[PalletIO6 6458], Comment=, ActivationMode=2, Cyclic=false
EventTableTriggerLogic 6455: layoutX=61, layoutY=50, Operand1=pallet3.2 6456, Operand2=pose3 6457, Operator=0, Delay=1000
EventTableTriggerIO 6456: IOValue=[-1], IRC5Controller=? -1, Operator=0, SignalSource=LCFA_profile 1
EventTableTriggerIO 6457: IOValue=[-1], IRC5Controller=? -1, Operator=0, SignalSource=LCFA_profile 1
EventTableActionIO 6458: IOValue=[-1], IRC5Controller=? -1, SignalTarget=LCFA_profile 1
EventTableEntry 6459: Group=, Trigger=AND 6460, Actions=[PalletIO7 6463], Comment=, ActivationMode=2, Cyclic=false
EventTableTriggerLogic 6460: layoutX=131, layoutY=52, Operand1=pickpallet1 6461, Operand2=pose7 6462, Operator=0, Delay=1000
EventTableTriggerIO 6461: IOValue=[-1], IRC5Controller=? -1, Operator=0, SignalSource=LCFA_profile 1
EventTableTriggerIO 6462: IOValue=[-1], IRC5Controller=? -1, Operator=0, SignalSource=LCFA_profile 1
EventTableActionIO 6463: IOValue=[-1], IRC5Controller=? -1, SignalTarget=LCFA_profile 1
EventTableEntry 6464: Group=, Trigger=AND 6465, Actions=[PalletIO8 6468], Comment=, ActivationMode=2, Cyclic=false
EventTableTriggerLogic 6465: layoutX=8, layoutY=16, Operand1=pickpallet2 6466, Operand2=pose13 6467, Operator=0, Delay=1000
EventTableTriggerIO 6466: IOValue=[-1], IRC5Controller=? -1, Operator=0, SignalSource=LCFA_profile 1
EventTableTriggerIO 6467: IOValue=[-1], IRC5Controller=? -1, Operator=0, SignalSource=LCFA_profile 1
EventTableActionIO 6468: IOValue=[-1], IRC5Controller=? -1, SignalTarget=LCFA_profile 1
EventTableEntry 6469: Group=, Trigger=AND 6470, Actions=[PalletIO9 6482], Comment=, ActivationMode=2, Cyclic=false
EventTableTriggerLogic 6470: layoutX=232, layoutY=117, Operand1=AND 6471, Operand2=pallet4 6481, Operator=0, Delay=1000
EventTableTriggerLogic 6471: layoutX=158, layoutY=65, Operand1=AND 6472, Operand2=AND 6477, Operator=0, Delay=1000
EventTableTriggerLogic 6472: layoutX=63, layoutY=28, Operand1=NOT 6473, Operand2=NOT 6475, Operator=0, Delay=1000
EventTableTriggerLogic 6473: layoutX=8, layoutY=16, Operand1=conv1_motor_s1 6474, Operand2=? -1, Operator=2, Delay=1000
EventTableTriggerIO 6474: IOValue=[-1], IRC5Controller=? -1, Operator=0, SignalSource=ALab_CellC_v1.0_4 5362
EventTableTriggerLogic 6475: layoutX=8, layoutY=52, Operand1=conv1_motor_s2 6476, Operand2=? -1, Operator=2, Delay=1000
EventTableTriggerIO 6476: IOValue=[-1], IRC5Controller=? -1, Operator=0, SignalSource=ALab_CellC_v1.0_4 5362
EventTableTriggerLogic 6477: layoutX=78, layoutY=103, Operand1=conv2_motor_s1 6478, Operand2=NOT 6479, Operator=0, Delay=1000
EventTableTriggerIO 6478: IOValue=[-1], IRC5Controller=? -1, Operator=0, SignalSource=ALab_CellC_v1.0_4 5362
EventTableTriggerLogic 6479: layoutX=6, layoutY=126, Operand1=conv2_motor_s2 6480, Operand2=? -1, Operator=2, Delay=1000
EventTableTriggerIO 6480: IOValue=[-1], IRC5Controller=? -1, Operator=0, SignalSource=ALab_CellC_v1.0_4 5362
EventTableTriggerIO 6481: IOValue=[-1], IRC5Controller=? -1, Operator=0, SignalSource=LCFA_profile 1
EventTableActionIO 6482: IOValue=[-1], IRC5Controller=? -1, SignalTarget=LCFA_profile 1
EventTableEntry 6483: Group=, Trigger=AND 6484, Actions=[PalletIO10 6493], Comment=, ActivationMode=2, Cyclic=false
EventTableTriggerLogic 6484: layoutX=237, layoutY=122, Operand1=AND 6485, Operand2=conv2_buffer_stopper 6492, Operator=0, Delay=1000
EventTableTriggerLogic 6485: layoutX=140, layoutY=22, Operand1=pallet4.1 6486, Operand2=AND 6487, Operator=0, Delay=1000
EventTableTriggerIO 6486: IOValue=[-1], IRC5Controller=? -1, Operator=0, SignalSource=LCFA_profile 1
EventTableTriggerLogic 6487: layoutX=90, layoutY=61, Operand1=cellC_pallet_holder 8127, Operand2=cellC_pallet_stopper 8128, Operator=0, Delay=1000
EventTableTriggerIO 6492: IOValue=[-1], IRC5Controller=? -1, Operator=0, SignalSource=ALab_CellC_v1.0_4 5362
EventTableActionIO 6493: IOValue=[-1], IRC5Controller=? -1, SignalTarget=LCFA_profile 1
EventTableEntry 6494: Group=, Trigger=AND 6495, Actions=[PalletIO11 6510], Comment=, ActivationMode=2, Cyclic=false
EventTableTriggerLogic 6495: layoutX=240, layoutY=90, Operand1=AND 6496, Operand2=AND 6500, Operator=0, Delay=1000
EventTableTriggerLogic 6496: layoutX=130, layoutY=37, Operand1=NOT 8011, Operand2=NOT 8013, Operator=0, Delay=1000
EventTableTriggerLogic 6500: layoutX=189, layoutY=138, Operand1=AND 6501, Operand2=AND 6506, Operator=0, Delay=1000
EventTableTriggerLogic 6501: layoutX=102, layoutY=97, Operand1=NOT 8015, Operand2=conv2_motor_s1 8017, Operator=0, Delay=1000
EventTableTriggerLogic 6506: layoutX=112, layoutY=167, Operand1=NOT 8018, Operand2=pallet5 8020, Operator=0, Delay=1000
EventTableActionIO 6510: IOValue=[-1], IRC5Controller=? -1, SignalTarget=LCFA_profile 1
EventTableEntry 6511: Group=, Trigger=AND 6512, Actions=[PalletIO12 6515], Comment=, ActivationMode=2, Cyclic=false
EventTableTriggerLogic 6512: layoutX=80, layoutY=49, Operand1=pallet5.1 6513, Operand2=conv2_outer_lifter 6514, Operator=0, Delay=1000
EventTableTriggerIO 6513: IOValue=[-1], IRC5Controller=? -1, Operator=0, SignalSource=LCFA_profile 1
EventTableTriggerIO 6514: IOValue=[-1], IRC5Controller=? -1, Operator=0, SignalSource=ALab_CellC_v1.0_4 5362
EventTableActionIO 6515: IOValue=[-1], IRC5Controller=? -1, SignalTarget=LCFA_profile 1
EventTableEntry 6516: Group=, Trigger=PalletIO1 6517, Actions=[pallet1 6518], Comment=, ActivationMode=2, Cyclic=false
EventTableTriggerIO 6517: IOValue=[1], IRC5Controller=? -1, Operator=0, SignalSource=LCFA_profile 1
EventTableActionIO 6518: IOValue=[1], IRC5Controller=? -1, SignalTarget=LCFA_profile 1
EventTableEntry 6519: Group=, Trigger=PalletIO2 6520, Actions=[pallet2 6521], Comment=, ActivationMode=2, Cyclic=false
EventTableTriggerIO 6520: IOValue=[1], IRC5Controller=? -1, Operator=0, SignalSource=LCFA_profile 1
EventTableActionIO 6521: IOValue=[1], IRC5Controller=? -1, SignalTarget=LCFA_profile 1
EventTableEntry 6525: Group=, Trigger=PalletIO4 6526, Actions=[pallet3 6527], Comment=, ActivationMode=2, Cyclic=false
EventTableTriggerIO 6526: IOValue=[1], IRC5Controller=? -1, Operator=0, SignalSource=LCFA_profile 1
EventTableActionIO 6527: IOValue=[1], IRC5Controller=? -1, SignalTarget=LCFA_profile 1
EventTableEntry 6528: Group=, Trigger=PalletIO5 6529, Actions=[pallet3.2 6530], Comment=, ActivationMode=2, Cyclic=false
EventTableTriggerIO 6529: IOValue=[1], IRC5Controller=? -1, Operator=0, SignalSource=LCFA_profile 1
EventTableActionIO 6530: IOValue=[1], IRC5Controller=? -1, SignalTarget=LCFA_profile 1
EventTableEntry 6531: Group=, Trigger=PalletIO6 6532, Actions=[pickpallet1 6533], Comment=, ActivationMode=2, Cyclic=false
EventTableTriggerIO 6532: IOValue=[1], IRC5Controller=? -1, Operator=0, SignalSource=LCFA_profile 1
EventTableActionIO 6533: IOValue=[1], IRC5Controller=? -1, SignalTarget=LCFA_profile 1
EventTableEntry 6534: Group=, Trigger=PalletIO7 6535, Actions=[pickpallet2 6536], Comment=, ActivationMode=2, Cyclic=false
EventTableTriggerIO 6535: IOValue=[1], IRC5Controller=? -1, Operator=0, SignalSource=LCFA_profile 1
EventTableActionIO 6536: IOValue=[1], IRC5Controller=? -1, SignalTarget=LCFA_profile 1
EventTableEntry 6537: Group=, Trigger=PalletIO8 6538, Actions=[pallet4 6539], Comment=, ActivationMode=2, Cyclic=false
EventTableTriggerIO 6538: IOValue=[1], IRC5Controller=? -1, Operator=0, SignalSource=LCFA_profile 1
EventTableActionIO 6539: IOValue=[1], IRC5Controller=? -1, SignalTarget=LCFA_profile 1
EventTableEntry 6540: Group=, Trigger=PalletIO9 6541, Actions=[pallet4.1 6542], Comment=, ActivationMode=2, Cyclic=false
EventTableTriggerIO 6541: IOValue=[1], IRC5Controller=? -1, Operator=0, SignalSource=LCFA_profile 1
EventTableActionIO 6542: IOValue=[1], IRC5Controller=? -1, SignalTarget=LCFA_profile 1
EventTableEntry 6543: Group=, Trigger=PalletIO10 6544, Actions=[pallet5 6545], Comment=, ActivationMode=2, Cyclic=false
EventTableTriggerIO 6544: IOValue=[1], IRC5Controller=? -1, Operator=0, SignalSource=LCFA_profile 1
EventTableActionIO 6545: IOValue=[1], IRC5Controller=? -1, SignalTarget=LCFA_profile 1
EventTableEntry 6546: Group=, Trigger=PalletIO11 6547, Actions=[pallet5.1 6548], Comment=, ActivationMode=2, Cyclic=false
EventTableTriggerIO 6547: IOValue=[1], IRC5Controller=? -1, Operator=0, SignalSource=LCFA_profile 1
EventTableActionIO 6548: IOValue=[1], IRC5Controller=? -1, SignalTarget=LCFA_profile 1
EventTableEntry 6555: Group=, Trigger=cellC_pallet_holder 6556, Actions=[cellC_pallet_holder_closed 6557], Comment=, ActivationMode=2, Cyclic=false
EventTableTriggerIO 6556: IOValue=[0], IRC5Controller=? -1, Operator=0, SignalSource=ALab_CellC_v1.0_4 5362
EventTableActionIO 6557: IOValue=[1], IRC5Controller=? -1, SignalTarget=ALab_CellC_v1.0_4 5362
EventTableEntry 6558: Group=, Trigger=cellC_pallet_holder 6559, Actions=[cellC_pallet_holder_closed 6560], Comment=, ActivationMode=2, Cyclic=false
EventTableTriggerIO 6559: IOValue=[1], IRC5Controller=? -1, Operator=0, SignalSource=ALab_CellC_v1.0_4 5362
EventTableActionIO 6560: IOValue=[0], IRC5Controller=? -1, SignalTarget=ALab_CellC_v1.0_4 5362
EventTableEntry 6561: Group=, Trigger=cellC_pallet_holder 6562, Actions=[cellC_pallet_holder_open 6563], Comment=, ActivationMode=2, Cyclic=false
EventTableTriggerIO 6562: IOValue=[0], IRC5Controller=? -1, Operator=0, SignalSource=ALab_CellC_v1.0_4 5362
EventTableActionIO 6563: IOValue=[0], IRC5Controller=? -1, SignalTarget=ALab_CellC_v1.0_4 5362
EventTableEntry 6564: Group=, Trigger=cellC_pallet_holder 6565, Actions=[cellC_pallet_holder_open 6566], Comment=, ActivationMode=2, Cyclic=false
EventTableTriggerIO 6565: IOValue=[1], IRC5Controller=? -1, Operator=0, SignalSource=ALab_CellC_v1.0_4 5362
EventTableActionIO 6566: IOValue=[1], IRC5Controller=? -1, SignalTarget=ALab_CellC_v1.0_4 5362
EventTableEntry 6567: Group=, Trigger=cellC_pallet_stopper 6568, Actions=[cellC_stopper_closed 6569], Comment=, ActivationMode=2, Cyclic=false
EventTableTriggerIO 6568: IOValue=[1], IRC5Controller=? -1, Operator=0, SignalSource=ALab_CellC_v1.0_4 5362
EventTableActionIO 6569: IOValue=[0], IRC5Controller=? -1, SignalTarget=ALab_CellC_v1.0_4 5362
EventTableEntry 6570: Group=, Trigger=cellC_pallet_stopper 6571, Actions=[cellC_stopper_closed 6572], Comment=, ActivationMode=2, Cyclic=false
EventTableTriggerIO 6571: IOValue=[0], IRC5Controller=? -1, Operator=0, SignalSource=ALab_CellC_v1.0_4 5362
EventTableActionIO 6572: IOValue=[1], IRC5Controller=? -1, SignalTarget=ALab_CellC_v1.0_4 5362
EventTableEntry 6573: Group=, Trigger=cellC_pallet_stopper 6574, Actions=[cellC_stopper_open 6575], Comment=, ActivationMode=2, Cyclic=false
EventTableTriggerIO 6574: IOValue=[0], IRC5Controller=? -1, Operator=0, SignalSource=ALab_CellC_v1.0_4 5362
EventTableActionIO 6575: IOValue=[0], IRC5Controller=? -1, SignalTarget=ALab_CellC_v1.0_4 5362
EventTableEntry 6576: Group=, Trigger=cellC_pallet_stopper 6577, Actions=[cellC_stopper_open 6578], Comment=, ActivationMode=2, Cyclic=false
EventTableTriggerIO 6577: IOValue=[1], IRC5Controller=? -1, Operator=0, SignalSource=ALab_CellC_v1.0_4 5362
EventTableActionIO 6578: IOValue=[1], IRC5Controller=? -1, SignalTarget=ALab_CellC_v1.0_4 5362
EventTableEntry 6579: Group=, Trigger=cellC_gripper_horizontal_move 6580, Actions=[cellC_gripper_horizontal_closed 6581], Comment=, ActivationMode=2, Cyclic=false
EventTableTriggerIO 6580: IOValue=[1], IRC5Controller=? -1, Operator=0, SignalSource=ALab_CellC_v1.0_4 5362
EventTableActionIO 6581: IOValue=[0], IRC5Controller=? -1, SignalTarget=ALab_CellC_v1.0_4 5362
EventTableEntry 6582: Group=, Trigger=cellC_gripper_horizontal_move 6583, Actions=[cellC_gripper_horizontal_closed 6584], Comment=, ActivationMode=2, Cyclic=false
EventTableTriggerIO 6583: IOValue=[0], IRC5Controller=? -1, Operator=0, SignalSource=ALab_CellC_v1.0_4 5362
EventTableActionIO 6584: IOValue=[1], IRC5Controller=? -1, SignalTarget=ALab_CellC_v1.0_4 5362
EventTableEntry 6585: Group=, Trigger=cellC_gripper_vertical_move 6586, Actions=[cellC_gripper_vertical_open 6587], Comment=, ActivationMode=2, Cyclic=false
EventTableTriggerIO 6586: IOValue=[1], IRC5Controller=? -1, Operator=0, SignalSource=ALab_CellC_v1.0_4 5362
EventTableActionIO 6587: IOValue=[1], IRC5Controller=? -1, SignalTarget=ALab_CellC_v1.0_4 5362
EventTableEntry 6588: Group=, Trigger=cellC_gripper_vertical_move 6589, Actions=[cellC_gripper_vertical_open 6590], Comment=, ActivationMode=2, Cyclic=false
EventTableTriggerIO 6589: IOValue=[0], IRC5Controller=? -1, Operator=0, SignalSource=ALab_CellC_v1.0_4 5362
EventTableActionIO 6590: IOValue=[0], IRC5Controller=? -1, SignalTarget=ALab_CellC_v1.0_4 5362
EventTableEntry 6591: Group=, Trigger=cellC_slider_vertical_move 6592, Actions=[cellC_slider_down 6593], Comment=, ActivationMode=2, Cyclic=false
EventTableTriggerIO 6592: IOValue=[0], IRC5Controller=? -1, Operator=0, SignalSource=ALab_CellC_v1.0_4 5362
EventTableActionIO 6593: IOValue=[0], IRC5Controller=? -1, SignalTarget=ALab_CellC_v1.0_4 5362
EventTableEntry 6594: Group=, Trigger=cellC_slider_vertical_move 6595, Actions=[cellC_slider_up 6596], Comment=, ActivationMode=2, Cyclic=false
EventTableTriggerIO 6595: IOValue=[1], IRC5Controller=? -1, Operator=0, SignalSource=ALab_CellC_v1.0_4 5362
EventTableActionIO 6596: IOValue=[0], IRC5Controller=? -1, SignalTarget=ALab_CellC_v1.0_4 5362
EventTableEntry 6597: Group=, Trigger=cellC_slider_vertical_move 6598, Actions=[cellC_slider_down 6599], Comment=, ActivationMode=2, Cyclic=false
EventTableTriggerIO 6598: IOValue=[1], IRC5Controller=? -1, Operator=0, SignalSource=ALab_CellC_v1.0_4 5362
EventTableActionIO 6599: IOValue=[1], IRC5Controller=? -1, SignalTarget=ALab_CellC_v1.0_4 5362
EventTableEntry 6600: Group=, Trigger=cellC_slider_vertical_move 6601, Actions=[cellC_slider_up 6602], Comment=, ActivationMode=2, Cyclic=false
EventTableTriggerIO 6601: IOValue=[0], IRC5Controller=? -1, Operator=0, SignalSource=ALab_CellC_v1.0_4 5362
EventTableActionIO 6602: IOValue=[1], IRC5Controller=? -1, SignalTarget=ALab_CellC_v1.0_4 5362
EventTableEntry 6603: Group=, Trigger=cellC_slider_horizontal_move 6604, Actions=[cellC_slider_over_conv1 6605], Comment=, ActivationMode=2, Cyclic=false
EventTableTriggerIO 6604: IOValue=[0], IRC5Controller=? -1, Operator=0, SignalSource=ALab_CellC_v1.0_4 5362
EventTableActionIO 6605: IOValue=[1], IRC5Controller=? -1, SignalTarget=ALab_CellC_v1.0_4 5362
EventTableEntry 6606: Group=, Trigger=cellC_slider_horizontal_move 6607, Actions=[cellC_slider_over_conv1 6608], Comment=, ActivationMode=2, Cyclic=false
EventTableTriggerIO 6607: IOValue=[1], IRC5Controller=? -1, Operator=0, SignalSource=ALab_CellC_v1.0_4 5362
EventTableActionIO 6608: IOValue=[0], IRC5Controller=? -1, SignalTarget=ALab_CellC_v1.0_4 5362
EventTableEntry 6609: Group=, Trigger=cellC_slider_horizontal_move 6610, Actions=[cellC_slider_over_conv2 6611], Comment=, ActivationMode=2, Cyclic=false
EventTableTriggerIO 6610: IOValue=[1], IRC5Controller=? -1, Operator=0, SignalSource=ALab_CellC_v1.0_4 5362
EventTableActionIO 6611: IOValue=[1], IRC5Controller=? -1, SignalTarget=ALab_CellC_v1.0_4 5362
EventTableEntry 6612: Group=, Trigger=cellC_slider_horizontal_move 6613, Actions=[cellC_slider_over_conv2 6614], Comment=, ActivationMode=2, Cyclic=false
EventTableTriggerIO 6613: IOValue=[0], IRC5Controller=? -1, Operator=0, SignalSource=ALab_CellC_v1.0_4 5362
EventTableActionIO 6614: IOValue=[0], IRC5Controller=? -1, SignalTarget=ALab_CellC_v1.0_4 5362
EventTableEntry 6615: Group=, Trigger=pallet3 6616, Actions=[cellC_pallet_conv1 6617], Comment=, ActivationMode=2, Cyclic=false
EventTableTriggerIO 6616: IOValue=[1], IRC5Controller=? -1, Operator=0, SignalSource=LCFA_profile 1
EventTableActionIO 6617: IOValue=[1], IRC5Controller=? -1, SignalTarget=ALab_CellC_v1.0_4 5362
EventTableEntry 6618: Group=, Trigger=pallet4 6619, Actions=[cellC_pallet_conv1 6620], Comment=, ActivationMode=2, Cyclic=false
EventTableTriggerIO 6619: IOValue=[1], IRC5Controller=? -1, Operator=0, SignalSource=LCFA_profile 1
EventTableActionIO 6620: IOValue=[0], IRC5Controller=? -1, SignalTarget=ALab_CellC_v1.0_4 5362
EventTableEntry 6621: Group=, Trigger=pallet4 6622, Actions=[cellC_pallet_conv2 6623], Comment=, ActivationMode=2, Cyclic=false
EventTableTriggerIO 6622: IOValue=[1], IRC5Controller=? -1, Operator=0, SignalSource=LCFA_profile 1
EventTableActionIO 6623: IOValue=[1], IRC5Controller=? -1, SignalTarget=ALab_CellC_v1.0_4 5362
EventTableEntry 6624: Group=, Trigger=pallet5 6625, Actions=[cellC_pallet_conv2 6626], Comment=, ActivationMode=2, Cyclic=false
EventTableTriggerIO 6625: IOValue=[1], IRC5Controller=? -1, Operator=0, SignalSource=LCFA_profile 1
EventTableActionIO 6626: IOValue=[0], IRC5Controller=? -1, SignalTarget=ALab_CellC_v1.0_4 5362
EventTableEntry 6627: Group=, Trigger=conv2_buffer_stopper 6628, Actions=[conv2_pallet_stopper_down 6629], Comment=, ActivationMode=2, Cyclic=false
EventTableTriggerIO 6628: IOValue=[1], IRC5Controller=? -1, Operator=0, SignalSource=ALab_CellC_v1.0_4 5362
EventTableActionIO 6629: IOValue=[0], IRC5Controller=? -1, SignalTarget=ALab_CellC_v1.0_4 5362
EventTableEntry 6630: Group=, Trigger=conv2_buffer_stopper 6631, Actions=[conv2_pallet_stopper_down 6632], Comment=, ActivationMode=2, Cyclic=false
EventTableTriggerIO 6631: IOValue=[0], IRC5Controller=? -1, Operator=0, SignalSource=ALab_CellC_v1.0_4 5362
EventTableActionIO 6632: IOValue=[1], IRC5Controller=? -1, SignalTarget=ALab_CellC_v1.0_4 5362
EventTableEntry 6633: Group=, Trigger=pallet1.1 6634, Actions=[conv1_pallet_out 6635], Comment=, ActivationMode=2, Cyclic=false
EventTableTriggerIO 6634: IOValue=[1], IRC5Controller=? -1, Operator=0, SignalSource=LCFA_profile 1
EventTableActionIO 6635: IOValue=[1], IRC5Controller=? -1, SignalTarget=ALab_CellC_v1.0_4 5362
EventTableEntry 6636: Group=, Trigger=pallet2 6637, Actions=[conv1_pallet_out 6638], Comment=, ActivationMode=2, Cyclic=false
EventTableTriggerIO 6637: IOValue=[1], IRC5Controller=? -1, Operator=0, SignalSource=LCFA_profile 1
EventTableActionIO 6638: IOValue=[0], IRC5Controller=? -1, SignalTarget=ALab_CellC_v1.0_4 5362
EventTableEntry 6639: Group=, Trigger=pallet6 6640, Actions=[conv2_pallet_out 6641], Comment=, ActivationMode=2, Cyclic=false
EventTableTriggerIO 6640: IOValue=[1], IRC5Controller=? -1, Operator=0, SignalSource=LCFA_profile 1
EventTableActionIO 6641: IOValue=[1], IRC5Controller=? -1, SignalTarget=ALab_CellC_v1.0_4 5362
EventTableEntry 6642: Group=, Trigger=pallet1.1 6643, Actions=[conv2_pallet_out 6644], Comment=, ActivationMode=2, Cyclic=false
EventTableTriggerIO 6643: IOValue=[1], IRC5Controller=? -1, Operator=0, SignalSource=LCFA_profile 1
EventTableActionIO 6644: IOValue=[0], IRC5Controller=? -1, SignalTarget=ALab_CellC_v1.0_4 5362
EventTableEntry 6645: Group=, Trigger=conv2_outer_lifter 6646, Actions=[conv2_outer_lifter_down 6647], Comment=, ActivationMode=2, Cyclic=false
EventTableTriggerIO 6646: IOValue=[1], IRC5Controller=? -1, Operator=0, SignalSource=ALab_CellC_v1.0_4 5362
EventTableActionIO 6647: IOValue=[1], IRC5Controller=? -1, SignalTarget=ALab_CellC_v1.0_4 5362
EventTableEntry 6648: Group=, Trigger=conv2_outer_lifter 6649, Actions=[conv2_outer_lifter_down 6650], Comment=, ActivationMode=2, Cyclic=false
EventTableTriggerIO 6649: IOValue=[0], IRC5Controller=? -1, Operator=0, SignalSource=ALab_CellC_v1.0_4 5362
EventTableActionIO 6650: IOValue=[0], IRC5Controller=? -1, SignalTarget=ALab_CellC_v1.0_4 5362
EventTableEntry 6651: Group=, Trigger=conv2_outer_lifter 6652, Actions=[conv2_outer_lifter_up 6653], Comment=, ActivationMode=2, Cyclic=false
EventTableTriggerIO 6652: IOValue=[1], IRC5Controller=? -1, Operator=0, SignalSource=ALab_CellC_v1.0_4 5362
EventTableActionIO 6653: IOValue=[0], IRC5Controller=? -1, SignalTarget=ALab_CellC_v1.0_4 5362
EventTableEntry 6654: Group=, Trigger=conv2_outer_lifter 6655, Actions=[conv2_outer_lifter_up 6656], Comment=, ActivationMode=2, Cyclic=false
EventTableTriggerIO 6655: IOValue=[0], IRC5Controller=? -1, Operator=0, SignalSource=ALab_CellC_v1.0_4 5362
EventTableActionIO 6656: IOValue=[1], IRC5Controller=? -1, SignalTarget=ALab_CellC_v1.0_4 5362
EventTableEntry 6657: Group=, Trigger=conv1_outer_lifter 6658, Actions=[conv1_outer_lifter_up 6659], Comment=, ActivationMode=2, Cyclic=false
EventTableTriggerIO 6658: IOValue=[0], IRC5Controller=? -1, Operator=0, SignalSource=ALab_CellC_v1.0_4 5362
EventTableActionIO 6659: IOValue=[1], IRC5Controller=? -1, SignalTarget=ALab_CellC_v1.0_4 5362
EventTableEntry 6660: Group=, Trigger=conv1_outer_lifter 6661, Actions=[conv1_outer_lifter_up 6662], Comment=, ActivationMode=2, Cyclic=false
EventTableTriggerIO 6661: IOValue=[1], IRC5Controller=? -1, Operator=0, SignalSource=ALab_CellC_v1.0_4 5362
EventTableActionIO 6662: IOValue=[0], IRC5Controller=? -1, SignalTarget=ALab_CellC_v1.0_4 5362
EventTableEntry 6663: Group=, Trigger=conv1_outer_lifter 6664, Actions=[conv1_outer_lifter_down 6665], Comment=, ActivationMode=2, Cyclic=false
EventTableTriggerIO 6664: IOValue=[1], IRC5Controller=? -1, Operator=0, SignalSource=ALab_CellC_v1.0_4 5362
EventTableActionIO 6665: IOValue=[1], IRC5Controller=? -1, SignalTarget=ALab_CellC_v1.0_4 5362
EventTableEntry 6666: Group=, Trigger=conv1_outer_lifter 6667, Actions=[conv1_outer_lifter_down 6668], Comment=, ActivationMode=2, Cyclic=false
EventTableTriggerIO 6667: IOValue=[0], IRC5Controller=? -1, Operator=0, SignalSource=ALab_CellC_v1.0_4 5362
EventTableActionIO 6668: IOValue=[0], IRC5Controller=? -1, SignalTarget=ALab_CellC_v1.0_4 5362
EventTableTriggerIO 6670: IOValue=[-1], IRC5Controller=? -1, Operator=0, SignalSource=ALab_CellC_v1.0_4 5362
EventTableTriggerIO 6671: IOValue=[-1], IRC5Controller=? -1, Operator=0, SignalSource=ALab_CellC_v1.0_4 5362
EventTableEntry 6694: Group=, Trigger=PalletIO3 6695, Actions=[pallet3.1 6696], Comment=, ActivationMode=2, Cyclic=false
EventTableTriggerIO 6695: IOValue=[1], IRC5Controller=? -1, Operator=0, SignalSource=LCFA_profile 1
EventTableActionIO 6696: IOValue=[1], IRC5Controller=? -1, SignalTarget=LCFA_profile 1
EventTableEntry 6700: Group=, Trigger=PalletIO12 6701, Actions=[pallet6 6702], Comment=, ActivationMode=2, Cyclic=false
EventTableTriggerIO 6701: IOValue=[1], IRC5Controller=? -1, Operator=0, SignalSource=LCFA_profile 1
EventTableActionIO 6702: IOValue=[1], IRC5Controller=? -1, SignalTarget=LCFA_profile 1
EventTableEntry 6703: Group=, Trigger=PalletIO13 6704, Actions=[pallet6.1 6705], Comment=, ActivationMode=2, Cyclic=false
EventTableTriggerIO 6704: IOValue=[1], IRC5Controller=? -1, Operator=0, SignalSource=LCFA_profile 1
EventTableActionIO 6705: IOValue=[1], IRC5Controller=? -1, SignalTarget=LCFA_profile 1
EventTableEntry 6706: Group=, Trigger=AND 6765, Actions=[PalletIO13 6707], Comment=, ActivationMode=2, Cyclic=false
EventTableActionIO 6707: IOValue=[-1], IRC5Controller=? -1, SignalTarget=LCFA_profile 1
EventTableEntry 6712: Group=, Trigger=pallet1.1 6713, Actions=[pallet1 6714], Comment=, ActivationMode=2, Cyclic=false
EventTableTriggerIO 6713: IOValue=[1], IRC5Controller=? -1, Operator=0, SignalSource=LCFA_profile 1
EventTableActionIO 6714: IOValue=[0], IRC5Controller=? -1, SignalTarget=LCFA_profile 1
EventTableEntry 6715: Group=, Trigger=pallet1.1 6716, Actions=[pallet2 6717], Comment=, ActivationMode=2, Cyclic=false
EventTableTriggerIO 6716: IOValue=[1], IRC5Controller=? -1, Operator=0, SignalSource=LCFA_profile 1
EventTableActionIO 6717: IOValue=[0], IRC5Controller=? -1, SignalTarget=LCFA_profile 1
EventTableEntry 6718: Group=, Trigger=pallet1.1 6719, Actions=[pallet3 6720], Comment=, ActivationMode=2, Cyclic=false
EventTableTriggerIO 6719: IOValue=[1], IRC5Controller=? -1, Operator=0, SignalSource=LCFA_profile 1
EventTableActionIO 6720: IOValue=[0], IRC5Controller=? -1, SignalTarget=LCFA_profile 1
EventTableEntry 6721: Group=, Trigger=pallet1.1 6722, Actions=[pallet3.1 6723], Comment=, ActivationMode=2, Cyclic=false
EventTableTriggerIO 6722: IOValue=[1], IRC5Controller=? -1, Operator=0, SignalSource=LCFA_profile 1
EventTableActionIO 6723: IOValue=[0], IRC5Controller=? -1, SignalTarget=LCFA_profile 1
EventTableEntry 6724: Group=, Trigger=pallet1.1 6725, Actions=[pallet3.2 6726], Comment=, ActivationMode=2, Cyclic=false
EventTableTriggerIO 6725: IOValue=[1], IRC5Controller=? -1, Operator=0, SignalSource=LCFA_profile 1
EventTableActionIO 6726: IOValue=[0], IRC5Controller=? -1, SignalTarget=LCFA_profile 1
EventTableEntry 6727: Group=, Trigger=pallet1.1 6728, Actions=[pickpallet1 6729], Comment=, ActivationMode=2, Cyclic=false
EventTableTriggerIO 6728: IOValue=[1], IRC5Controller=? -1, Operator=0, SignalSource=LCFA_profile 1
EventTableActionIO 6729: IOValue=[0], IRC5Controller=? -1, SignalTarget=LCFA_profile 1
EventTableEntry 6730: Group=, Trigger=pallet1.1 6731, Actions=[pickpallet2 6732], Comment=, ActivationMode=2, Cyclic=false
EventTableTriggerIO 6731: IOValue=[1], IRC5Controller=? -1, Operator=0, SignalSource=LCFA_profile 1
EventTableActionIO 6732: IOValue=[0], IRC5Controller=? -1, SignalTarget=LCFA_profile 1
EventTableEntry 6733: Group=, Trigger=pallet1.1 6734, Actions=[pallet4 6735], Comment=, ActivationMode=2, Cyclic=false
EventTableTriggerIO 6734: IOValue=[1], IRC5Controller=? -1, Operator=0, SignalSource=LCFA_profile 1
EventTableActionIO 6735: IOValue=[0], IRC5Controller=? -1, SignalTarget=LCFA_profile 1
EventTableEntry 6736: Group=, Trigger=pallet1.1 6737, Actions=[pallet4.1 6738], Comment=, ActivationMode=2, Cyclic=false
EventTableTriggerIO 6737: IOValue=[1], IRC5Controller=? -1, Operator=0, SignalSource=LCFA_profile 1
EventTableActionIO 6738: IOValue=[0], IRC5Controller=? -1, SignalTarget=LCFA_profile 1
EventTableEntry 6739: Group=, Trigger=pallet1.1 6740, Actions=[pallet5 6741], Comment=, ActivationMode=2, Cyclic=false
EventTableTriggerIO 6740: IOValue=[1], IRC5Controller=? -1, Operator=0, SignalSource=LCFA_profile 1
EventTableActionIO 6741: IOValue=[0], IRC5Controller=? -1, SignalTarget=LCFA_profile 1
EventTableEntry 6742: Group=, Trigger=pallet1.1 6743, Actions=[pallet5.1 6744], Comment=, ActivationMode=2, Cyclic=false
EventTableTriggerIO 6743: IOValue=[1], IRC5Controller=? -1, Operator=0, SignalSource=LCFA_profile 1
EventTableActionIO 6744: IOValue=[0], IRC5Controller=? -1, SignalTarget=LCFA_profile 1
EventTableEntry 6745: Group=, Trigger=pallet1.1 6746, Actions=[pallet6 6747], Comment=, ActivationMode=2, Cyclic=false
EventTableTriggerIO 6746: IOValue=[1], IRC5Controller=? -1, Operator=0, SignalSource=LCFA_profile 1
EventTableActionIO 6747: IOValue=[0], IRC5Controller=? -1, SignalTarget=LCFA_profile 1
EventTableEntry 6748: Group=, Trigger=AND 6750, Actions=[PalletIO14 6749], Comment=, ActivationMode=2, Cyclic=false
EventTableActionIO 6749: IOValue=[-1], IRC5Controller=? -1, SignalTarget=LCFA_profile 1
EventTableTriggerLogic 6750: layoutX=155, layoutY=137, Operand1=AND 6751, Operand2=NOT 6755, Operator=0, Delay=1000
EventTableTriggerLogic 6751: layoutX=117, layoutY=11, Operand1=pallet6.1 6752, Operand2=NOT 6763, Operator=0, Delay=1000
EventTableTriggerIO 6752: IOValue=[-1], IRC5Controller=? -1, Operator=0, SignalSource=LCFA_profile 1
EventTableTriggerLogic 6755: layoutX=8, layoutY=81, Operand1=conv2_motor_s1 6774, Operand2=? -1, Operator=2, Delay=1000
EventTableEntry 6760: Group=, Trigger=PalletIO14 6761, Actions=[pallet1.1 6762], Comment=, ActivationMode=2, Cyclic=false
EventTableTriggerIO 6761: IOValue=[1], IRC5Controller=? -1, Operator=0, SignalSource=LCFA_profile 1
EventTableActionIO 6762: IOValue=[1], IRC5Controller=? -1, SignalTarget=LCFA_profile 1
EventTableTriggerLogic 6763: layoutX=20, layoutY=39, Operand1=conv1_outer_lifter 6764, Operand2=? -1, Operator=2, Delay=1000
EventTableTriggerIO 6764: IOValue=[-1], IRC5Controller=? -1, Operator=0, SignalSource=ALab_CellC_v1.0_4 5362
EventTableTriggerLogic 6765: layoutX=150, layoutY=90, Operand1=AND 6770, Operand2=conv2_motor_s1 6766, Operator=0, Delay=1000
EventTableTriggerIO 6766: IOValue=[-1], IRC5Controller=? -1, Operator=0, SignalSource=ALab_CellC_v1.0_4 5362
EventTableEntry 6767: Group=, Trigger=pallet1.1 6768, Actions=[pallet6.1 6769], Comment=, ActivationMode=2, Cyclic=false
EventTableTriggerIO 6768: IOValue=[1], IRC5Controller=? -1, Operator=0, SignalSource=LCFA_profile 1
EventTableActionIO 6769: IOValue=[0], IRC5Controller=? -1, SignalTarget=LCFA_profile 1
EventTableTriggerLogic 6770: layoutX=62, layoutY=30, Operand1=pallet6 6771, Operand2=NOT 6772, Operator=0, Delay=1000
EventTableTriggerIO 6771: IOValue=[-1], IRC5Controller=? -1, Operator=0, SignalSource=LCFA_profile 1
EventTableTriggerLogic 6772: layoutX=10, layoutY=51, Operand1=conv2_outer_lifter 6773, Operand2=? -1, Operator=2, Delay=1000
EventTableTriggerIO 6773: IOValue=[-1], IRC5Controller=? -1, Operator=0, SignalSource=ALab_CellC_v1.0_4 5362
EventTableTriggerIO 6774: IOValue=[-1], IRC5Controller=? -1, Operator=0, SignalSource=ALab_CellC_v1.0_4 5362
EventTableEntry 6775: Group=, Trigger=AND 6777, Actions=[PalletIO1 6776], Comment=, ActivationMode=2, Cyclic=false
EventTableActionIO 6776: IOValue=[-1], IRC5Controller=? -1, SignalTarget=LCFA_profile 1
EventTableTriggerLogic 6777: layoutX=48, layoutY=41, Operand1=pallet1.1 6778, Operand2=PalletIO00 6779, Operator=0, Delay=1000
EventTableTriggerIO 6778: IOValue=[-1], IRC5Controller=? -1, Operator=0, SignalSource=LCFA_profile 1
EventTableTriggerIO 6779: IOValue=[-1], IRC5Controller=? -1, Operator=0, SignalSource=LCFA_profile 1
EventTableEntry 6780: Group=, Trigger=pallet1 6781, Actions=[pallet1.1 6782], Comment=, ActivationMode=2, Cyclic=false
EventTableTriggerIO 6781: IOValue=[1], IRC5Controller=? -1, Operator=0, SignalSource=LCFA_profile 1
EventTableActionIO 6782: IOValue=[0], IRC5Controller=? -1, SignalTarget=LCFA_profile 1
EventTableEntry 6783: Group=, Trigger=conv2_buffer_stopper 6784, Actions=[conv2_pallet_stopper_up 6785], Comment=, ActivationMode=2, Cyclic=false
EventTableTriggerIO 6784: IOValue=[1], IRC5Controller=? -1, Operator=0, SignalSource=ALab_CellC_v1.0_4 5362
EventTableActionIO 6785: IOValue=[1], IRC5Controller=? -1, SignalTarget=ALab_CellC_v1.0_4 5362
EventTableEntry 6786: Group=, Trigger=conv2_buffer_stopper 6787, Actions=[conv2_pallet_stopper_up 6788], Comment=, ActivationMode=2, Cyclic=false
EventTableTriggerIO 6787: IOValue=[0], IRC5Controller=? -1, Operator=0, SignalSource=ALab_CellC_v1.0_4 5362
EventTableActionIO 6788: IOValue=[0], IRC5Controller=? -1, SignalTarget=ALab_CellC_v1.0_4 5362
EventTableTriggerIO 7096: IOValue=[-1], IRC5Controller=? -1, Operator=0, SignalSource=ALab_CellC_v1.0_4 5362
EventTableTriggerIO 7097: IOValue=[-1], IRC5Controller=? -1, Operator=0, SignalSource=ALab_CellC_v1.0_4 5362
EventTableTriggerIO 7098: IOValue=[-1], IRC5Controller=? -1, Operator=0, SignalSource=ALab_CellC_v1.0_4 5362
EventTableTriggerIO 7099: IOValue=[-1], IRC5Controller=? -1, Operator=0, SignalSource=ALab_CellC_v1.0_4 5362
EventTableTriggerIO 7100: IOValue=[-1], IRC5Controller=? -1, Operator=0, SignalSource=ALab_CellC_v1.0_4 5362
EventTableTriggerIO 7101: IOValue=[-1], IRC5Controller=? -1, Operator=0, SignalSource=ALab_CellC_v1.0_4 5362
EventTableTriggerIO 7102: IOValue=[-1], IRC5Controller=? -1, Operator=0, SignalSource=ALab_CellC_v1.0_4 5362
EventTableTriggerIO 7103: IOValue=[-1], IRC5Controller=? -1, Operator=0, SignalSource=ALab_CellC_v1.0_4 5362
EventTableTriggerLogic 7105: layoutX=39, layoutY=51, Operand1=cellC_gripper_vertical_move 7959, Operand2=? -1, Operator=2, Delay=1000
EventTableTriggerIO 7106: IOValue=[-1], IRC5Controller=? -1, Operator=0, SignalSource=ALab_CellC_v1.0_4 5362
EventTableTriggerLogic 7107: layoutX=18, layoutY=53, Operand1=cellC_gripper_vertical_move 7108, Operand2=? -1, Operator=2, Delay=1000
EventTableTriggerIO 7108: IOValue=[-1], IRC5Controller=? -1, Operator=0, SignalSource=ALab_CellC_v1.0_4 5362
EventTableTriggerLogic 7110: layoutX=24, layoutY=52, Operand1=cellC_gripper_vertical_move 7963, Operand2=? -1, Operator=2, Delay=1000
EventTableTriggerLogic 7112: layoutX=34, layoutY=52, Operand1=cellC_gripper_vertical_move 7967, Operand2=? -1, Operator=2, Delay=1000
EventTableTriggerLogic 7117: layoutX=8, layoutY=16, Operand1=cellC_gripper_horizontal_move 7987, Operand2=? -1, Operator=2, Delay=1000
EventTableTriggerLogic 7118: layoutX=29, layoutY=45, Operand1=cellC_gripper_vertical_move 7988, Operand2=? -1, Operator=2, Delay=1000
EventTableTriggerLogic 7119: layoutX=8, layoutY=16, Operand1=cellC_gripper_horizontal_move 7991, Operand2=? -1, Operator=2, Delay=1000
EventTableTriggerLogic 7120: layoutX=23, layoutY=54, Operand1=cellC_gripper_vertical_move 7992, Operand2=? -1, Operator=2, Delay=1000
EventTableTriggerLogic 7121: layoutX=8, layoutY=16, Operand1=cellC_gripper_horizontal_move 7995, Operand2=? -1, Operator=2, Delay=1000
EventTableTriggerLogic 7122: layoutX=21, layoutY=52, Operand1=cellC_gripper_vertical_move 7996, Operand2=? -1, Operator=2, Delay=1000
EventTableTriggerLogic 7123: layoutX=8, layoutY=16, Operand1=cellC_gripper_horizontal_move 7999, Operand2=? -1, Operator=2, Delay=1000
EventTableTriggerLogic 7124: layoutX=15, layoutY=56, Operand1=cellC_gripper_vertical_move 8000, Operand2=? -1, Operator=2, Delay=1000
EventTableTriggerIO 7125: IOValue=[-1], IRC5Controller=? -1, Operator=0, SignalSource=ALab_CellC_v1.0_4 5362
EventTableTriggerIO 7126: IOValue=[-1], IRC5Controller=? -1, Operator=0, SignalSource=ALab_CellC_v1.0_4 5362
EventTableTriggerIO 7127: IOValue=[-1], IRC5Controller=? -1, Operator=0, SignalSource=ALab_CellC_v1.0_4 5362
EventTableTriggerLogic 7128: layoutX=45, layoutY=22, Operand1=cellC_pallet_holder 7129, Operand2=? -1, Operator=2, Delay=1000
EventTableTriggerIO 7129: IOValue=[-1], IRC5Controller=? -1, Operator=0, SignalSource=ALab_CellC_v1.0_4 5362
EventTableTriggerLogic 7130: layoutX=8, layoutY=16, Operand1=cellC_pallet_holder 7131, Operand2=? -1, Operator=2, Delay=1000
EventTableTriggerIO 7131: IOValue=[-1], IRC5Controller=? -1, Operator=0, SignalSource=ALab_CellC_v1.0_4 5362
EventTableTriggerLogic 7132: layoutX=12, layoutY=65, Operand1=cellC_pallet_stopper 7133, Operand2=? -1, Operator=2, Delay=1000
EventTableTriggerIO 7133: IOValue=[-1], IRC5Controller=? -1, Operator=0, SignalSource=ALab_CellC_v1.0_4 5362
EventTableTriggerIO 7134: IOValue=[-1], IRC5Controller=? -1, Operator=0, SignalSource=ALab_CellC_v1.0_4 5362
EventTableTriggerLogic 7135: layoutX=19, layoutY=95, Operand1=cellC_pallet_stopper 7136, Operand2=? -1, Operator=2, Delay=1000
EventTableTriggerIO 7136: IOValue=[-1], IRC5Controller=? -1, Operator=0, SignalSource=ALab_CellC_v1.0_4 5362
EventTableTriggerIO 7959: IOValue=[-1], IRC5Controller=? -1, Operator=0, SignalSource=ALab_CellC_v1.0_4 5362
EventTableTriggerIO 7960: IOValue=[-1], IRC5Controller=? -1, Operator=0, SignalSource=ALab_CellC_v1.0_4 5362
EventTableTriggerIO 7961: IOValue=[-1], IRC5Controller=? -1, Operator=0, SignalSource=ALab_CellC_v1.0_4 5362
EventTableTriggerIO 7962: IOValue=[-1], IRC5Controller=? -1, Operator=0, SignalSource=ALab_CellC_v1.0_4 5362
EventTableTriggerIO 7963: IOValue=[-1], IRC5Controller=? -1, Operator=0, SignalSource=ALab_CellC_v1.0_4 5362
EventTableTriggerIO 7964: IOValue=[-1], IRC5Controller=? -1, Operator=0, SignalSource=ALab_CellC_v1.0_4 5362
EventTableTriggerIO 7965: IOValue=[-1], IRC5Controller=? -1, Operator=0, SignalSource=ALab_CellC_v1.0_4 5362
EventTableTriggerIO 7966: IOValue=[-1], IRC5Controller=? -1, Operator=0, SignalSource=ALab_CellC_v1.0_4 5362
EventTableTriggerIO 7967: IOValue=[-1], IRC5Controller=? -1, Operator=0, SignalSource=ALab_CellC_v1.0_4 5362
EventTableTriggerIO 7968: IOValue=[-1], IRC5Controller=? -1, Operator=0, SignalSource=ALab_CellC_v1.0_4 5362
EventTableTriggerIO 7969: IOValue=[-1], IRC5Controller=? -1, Operator=0, SignalSource=ALab_CellC_v1.0_4 5362
EventTableTriggerIO 7970: IOValue=[-1], IRC5Controller=? -1, Operator=0, SignalSource=ALab_CellC_v1.0_4 5362
EventTableTriggerIO 7972: IOValue=[-1], IRC5Controller=? -1, Operator=0, SignalSource=ALab_CellC_v1.0_4 5362
EventTableTriggerIO 7973: IOValue=[-1], IRC5Controller=? -1, Operator=0, SignalSource=ALab_CellC_v1.0_4 5362
EventTableTriggerIO 7974: IOValue=[-1], IRC5Controller=? -1, Operator=0, SignalSource=ALab_CellC_v1.0_4 5362
EventTableTriggerIO 7976: IOValue=[-1], IRC5Controller=? -1, Operator=0, SignalSource=ALab_CellC_v1.0_4 5362
EventTableTriggerIO 7977: IOValue=[-1], IRC5Controller=? -1, Operator=0, SignalSource=ALab_CellC_v1.0_4 5362
EventTableTriggerIO 7978: IOValue=[-1], IRC5Controller=? -1, Operator=0, SignalSource=ALab_CellC_v1.0_4 5362
EventTableTriggerIO 7980: IOValue=[-1], IRC5Controller=? -1, Operator=0, SignalSource=ALab_CellC_v1.0_4 5362
EventTableTriggerIO 7981: IOValue=[-1], IRC5Controller=? -1, Operator=0, SignalSource=ALab_CellC_v1.0_4 5362
EventTableTriggerIO 7982: IOValue=[-1], IRC5Controller=? -1, Operator=0, SignalSource=ALab_CellC_v1.0_4 5362
EventTableTriggerIO 7984: IOValue=[-1], IRC5Controller=? -1, Operator=0, SignalSource=ALab_CellC_v1.0_4 5362
EventTableTriggerIO 7985: IOValue=[-1], IRC5Controller=? -1, Operator=0, SignalSource=ALab_CellC_v1.0_4 5362
EventTableTriggerIO 7986: IOValue=[-1], IRC5Controller=? -1, Operator=0, SignalSource=ALab_CellC_v1.0_4 5362
EventTableTriggerIO 7987: IOValue=[-1], IRC5Controller=? -1, Operator=0, SignalSource=ALab_CellC_v1.0_4 5362
EventTableTriggerIO 7988: IOValue=[-1], IRC5Controller=? -1, Operator=0, SignalSource=ALab_CellC_v1.0_4 5362
EventTableTriggerIO 7989: IOValue=[-1], IRC5Controller=? -1, Operator=0, SignalSource=ALab_CellC_v1.0_4 5362
EventTableTriggerIO 7990: IOValue=[-1], IRC5Controller=? -1, Operator=0, SignalSource=ALab_CellC_v1.0_4 5362
EventTableTriggerIO 7991: IOValue=[-1], IRC5Controller=? -1, Operator=0, SignalSource=ALab_CellC_v1.0_4 5362
EventTableTriggerIO 7992: IOValue=[-1], IRC5Controller=? -1, Operator=0, SignalSource=ALab_CellC_v1.0_4 5362
EventTableTriggerIO 7993: IOValue=[-1], IRC5Controller=? -1, Operator=0, SignalSource=ALab_CellC_v1.0_4 5362
EventTableTriggerIO 7994: IOValue=[-1], IRC5Controller=? -1, Operator=0, SignalSource=ALab_CellC_v1.0_4 5362
EventTableTriggerIO 7995: IOValue=[-1], IRC5Controller=? -1, Operator=0, SignalSource=ALab_CellC_v1.0_4 5362
EventTableTriggerIO 7996: IOValue=[-1], IRC5Controller=? -1, Operator=0, SignalSource=ALab_CellC_v1.0_4 5362
EventTableTriggerIO 7997: IOValue=[-1], IRC5Controller=? -1, Operator=0, SignalSource=ALab_CellC_v1.0_4 5362
EventTableTriggerIO 7998: IOValue=[-1], IRC5Controller=? -1, Operator=0, SignalSource=ALab_CellC_v1.0_4 5362
EventTableTriggerIO 7999: IOValue=[-1], IRC5Controller=? -1, Operator=0, SignalSource=ALab_CellC_v1.0_4 5362
EventTableTriggerIO 8000: IOValue=[-1], IRC5Controller=? -1, Operator=0, SignalSource=ALab_CellC_v1.0_4 5362
EventTableTriggerIO 8001: IOValue=[-1], IRC5Controller=? -1, Operator=0, SignalSource=ALab_CellC_v1.0_4 5362
EventTableTriggerIO 8002: IOValue=[-1], IRC5Controller=? -1, Operator=0, SignalSource=ALab_CellC_v1.0_4 5362
EventTableTriggerLogic 8003: layoutX=13, layoutY=13, Operand1=cellC_gripper_horizontal_move 8004, Operand2=? -1, Operator=2, Delay=1000
EventTableTriggerIO 8004: IOValue=[-1], IRC5Controller=? -1, Operator=0, SignalSource=ALab_CellC_v1.0_4 5362
EventTableTriggerLogic 8005: layoutX=36, layoutY=17, Operand1=cellC_gripper_horizontal_move 8006, Operand2=? -1, Operator=2, Delay=1000
EventTableTriggerIO 8006: IOValue=[-1], IRC5Controller=? -1, Operator=0, SignalSource=ALab_CellC_v1.0_4 5362
EventTableTriggerLogic 8007: layoutX=8, layoutY=16, Operand1=cellC_gripper_horizontal_move 8008, Operand2=? -1, Operator=2, Delay=1000
EventTableTriggerIO 8008: IOValue=[-1], IRC5Controller=? -1, Operator=0, SignalSource=ALab_CellC_v1.0_4 5362
EventTableTriggerLogic 8009: layoutX=8, layoutY=16, Operand1=cellC_gripper_horizontal_move 8010, Operand2=? -1, Operator=2, Delay=1000
EventTableTriggerIO 8010: IOValue=[-1], IRC5Controller=? -1, Operator=0, SignalSource=ALab_CellC_v1.0_4 5362
EventTableTriggerLogic 8011: layoutX=28, layoutY=18, Operand1=conv2_buffer_stopper 8012, Operand2=? -1, Operator=2, Delay=1000
EventTableTriggerIO 8012: IOValue=[-1], IRC5Controller=? -1, Operator=0, SignalSource=ALab_CellC_v1.0_4 5362
EventTableTriggerLogic 8013: layoutX=31, layoutY=56, Operand1=conv1_motor_s1 8014, Operand2=? -1, Operator=2, Delay=1000
EventTableTriggerIO 8014: IOValue=[-1], IRC5Controller=? -1, Operator=0, SignalSource=ALab_CellC_v1.0_4 5362
EventTableTriggerLogic 8015: layoutX=26, layoutY=90, Operand1=conv1_motor_s2 8016, Operand2=? -1, Operator=2, Delay=1000
EventTableTriggerIO 8016: IOValue=[-1], IRC5Controller=? -1, Operator=0, SignalSource=ALab_CellC_v1.0_4 5362
EventTableTriggerIO 8017: IOValue=[-1], IRC5Controller=? -1, Operator=0, SignalSource=ALab_CellC_v1.0_4 5362
EventTableTriggerLogic 8018: layoutX=29, layoutY=147, Operand1=conv2_motor_s2 8019, Operand2=? -1, Operator=2, Delay=1000
EventTableTriggerIO 8019: IOValue=[-1], IRC5Controller=? -1, Operator=0, SignalSource=ALab_CellC_v1.0_4 5362
EventTableTriggerIO 8020: IOValue=[-1], IRC5Controller=? -1, Operator=0, SignalSource=LCFA_profile 1
EventTableEntry 8024: Group=, Trigger=AND 8025, Actions=[PalletIO16 8026], Comment=, ActivationMode=2, Cyclic=false
EventTableTriggerLogic 8025: layoutX=103, layoutY=47, Operand1=NOT 8291, Operand2=pallet5 8290, Operator=0, Delay=1000
EventTableActionIO 8026: IOValue=[-1], IRC5Controller=? -1, SignalTarget=LCFA_profile 1
EventTableEntry 8027: Group=, Trigger=AND 8028, Actions=[PalletIO17 8032], Comment=, ActivationMode=2, Cyclic=false
EventTableTriggerLogic 8028: layoutX=79, layoutY=37, Operand1=Pallet5.3 8029, Operand2=conv2_buffer_upper_vertical_move 8133, Operator=0, Delay=1000
EventTableTriggerIO 8029: IOValue=[-1], IRC5Controller=? -1, Operator=0, SignalSource=LCFA_profile 1
EventTableActionIO 8032: IOValue=[-1], IRC5Controller=? -1, SignalTarget=LCFA_profile 1
EventTableEntry 8033: Group=, Trigger=AND 8034, Actions=[PalletIO19 8037], Comment=, ActivationMode=2, Cyclic=false
EventTableTriggerLogic 8034: layoutX=40, layoutY=37, Operand1=Pallet5.4 8035, Operand2=conv2_buffer_lower_vertical_move 8036, Operator=0, Delay=1000
EventTableTriggerIO 8035: IOValue=[-1], IRC5Controller=? -1, Operator=0, SignalSource=LCFA_profile 1
EventTableTriggerIO 8036: IOValue=[-1], IRC5Controller=? -1, Operator=0, SignalSource=ALab_CellC_v1.0_4 5362
EventTableActionIO 8037: IOValue=[-1], IRC5Controller=? -1, SignalTarget=LCFA_profile 1
EventTableEntry 8038: Group=, Trigger=AND 8039, Actions=[PalletIO22 8043], Comment=, ActivationMode=2, Cyclic=false
EventTableTriggerLogic 8039: layoutX=103, layoutY=47, Operand1=conv2_buffer_horizontal_move 8134, Operand2=Pallet5.7 8040, Operator=0, Delay=1000
EventTableTriggerIO 8040: IOValue=[-1], IRC5Controller=? -1, Operator=0, SignalSource=LCFA_profile 1
EventTableActionIO 8043: IOValue=[-1], IRC5Controller=? -1, SignalTarget=LCFA_profile 1
EventTableEntry 8044: Group=, Trigger=AND 8045, Actions=[PalletIO21 8048], Comment=, ActivationMode=2, Cyclic=false
EventTableTriggerLogic 8045: layoutX=54, layoutY=45, Operand1=NOT 8135, Operand2=Pallet5.6 8046, Operator=0, Delay=1000
EventTableTriggerIO 8046: IOValue=[-1], IRC5Controller=? -1, Operator=0, SignalSource=LCFA_profile 1
EventTableActionIO 8048: IOValue=[-1], IRC5Controller=? -1, SignalTarget=LCFA_profile 1
EventTableEntry 8049: Group=, Trigger=AND 8050, Actions=[PalletIO20 8054], Comment=, ActivationMode=2, Cyclic=false
EventTableTriggerLogic 8050: layoutX=108, layoutY=46, Operand1=NOT 8052, Operand2=Pallet5.5 8051, Operator=0, Delay=1000
EventTableTriggerIO 8051: IOValue=[-1], IRC5Controller=? -1, Operator=0, SignalSource=LCFA_profile 1
EventTableTriggerLogic 8052: layoutX=42, layoutY=19, Operand1=conv2_buffer_lower_vertical_move 8053, Operand2=? -1, Operator=2, Delay=1000
EventTableTriggerIO 8053: IOValue=[-1], IRC5Controller=? -1, Operator=0, SignalSource=ALab_CellC_v1.0_4 5362
EventTableActionIO 8054: IOValue=[-1], IRC5Controller=? -1, SignalTarget=LCFA_profile 1
EventTableEntry 8062: Group=, Trigger=PalletIO16 8063, Actions=[Pallet5.3 8064], Comment=, ActivationMode=2, Cyclic=false
EventTableTriggerIO 8063: IOValue=[1], IRC5Controller=? -1, Operator=0, SignalSource=LCFA_profile 1
EventTableActionIO 8064: IOValue=[1], IRC5Controller=? -1, SignalTarget=LCFA_profile 1
EventTableEntry 8065: Group=, Trigger=PalletIO17 8066, Actions=[Pallet5.4 8067], Comment=, ActivationMode=2, Cyclic=false
EventTableTriggerIO 8066: IOValue=[1], IRC5Controller=? -1, Operator=0, SignalSource=LCFA_profile 1
EventTableActionIO 8067: IOValue=[1], IRC5Controller=? -1, SignalTarget=LCFA_profile 1
EventTableEntry 8068: Group=, Trigger=PalletIO19 8069, Actions=[Pallet5.5 8070], Comment=, ActivationMode=2, Cyclic=false
EventTableTriggerIO 8069: IOValue=[1], IRC5Controller=? -1, Operator=0, SignalSource=LCFA_profile 1
EventTableActionIO 8070: IOValue=[1], IRC5Controller=? -1, SignalTarget=LCFA_profile 1
EventTableEntry 8071: Group=, Trigger=PalletIO20 8072, Actions=[Pallet5.6 8073], Comment=, ActivationMode=2, Cyclic=false
EventTableTriggerIO 8072: IOValue=[1], IRC5Controller=? -1, Operator=0, SignalSource=LCFA_profile 1
EventTableActionIO 8073: IOValue=[1], IRC5Controller=? -1, SignalTarget=LCFA_profile 1
EventTableEntry 8074: Group=, Trigger=PalletIO21 8075, Actions=[Pallet5.7 8076], Comment=, ActivationMode=2, Cyclic=false
EventTableTriggerIO 8075: IOValue=[1], IRC5Controller=? -1, Operator=0, SignalSource=LCFA_profile 1
EventTableActionIO 8076: IOValue=[1], IRC5Controller=? -1, SignalTarget=LCFA_profile 1
EventTableEntry 8077: Group=, Trigger=PalletIO22 8078, Actions=[Pallet5.8 8079], Comment=, ActivationMode=2, Cyclic=false
EventTableTriggerIO 8078: IOValue=[1], IRC5Controller=? -1, Operator=0, SignalSource=LCFA_profile 1
EventTableActionIO 8079: IOValue=[1], IRC5Controller=? -1, SignalTarget=LCFA_profile 1
EventTableEntry 8080: Group=, Trigger=Pallet5.3 8081, Actions=[pallet5 8082], Comment=, ActivationMode=2, Cyclic=false
EventTableTriggerIO 8081: IOValue=[1], IRC5Controller=? -1, Operator=0, SignalSource=LCFA_profile 1
EventTableActionIO 8082: IOValue=[0], IRC5Controller=? -1, SignalTarget=LCFA_profile 1
EventTableEntry 8083: Group=, Trigger=Pallet5.5 8084, Actions=[pickpallet3 8085], Comment=, ActivationMode=2, Cyclic=false
EventTableTriggerIO 8084: IOValue=[1], IRC5Controller=? -1, Operator=0, SignalSource=LCFA_profile 1
EventTableActionIO 8085: IOValue=[1], IRC5Controller=? -1, SignalTarget=LCFA_profile 1
EventTableEntry 8086: Group=, Trigger=Pallet5.8 8087, Actions=[pallet5 8088], Comment=, ActivationMode=2, Cyclic=false
EventTableTriggerIO 8087: IOValue=[1], IRC5Controller=? -1, Operator=0, SignalSource=LCFA_profile 1
EventTableActionIO 8088: IOValue=[1], IRC5Controller=? -1, SignalTarget=LCFA_profile 1
EventTableEntry 8089: Group=, Trigger=Pallet5.8 8090, Actions=[pickpallet3 8091], Comment=, ActivationMode=2, Cyclic=false
EventTableTriggerIO 8090: IOValue=[1], IRC5Controller=? -1, Operator=0, SignalSource=LCFA_profile 1
EventTableActionIO 8091: IOValue=[0], IRC5Controller=? -1, SignalTarget=LCFA_profile 1
EventTableEntry 8092: Group=, Trigger=pallet1.1 8093, Actions=[Pallet5.2 8094], Comment=, ActivationMode=2, Cyclic=false
EventTableTriggerIO 8093: IOValue=[1], IRC5Controller=? -1, Operator=0, SignalSource=LCFA_profile 1
EventTableActionIO 8094: IOValue=[0], IRC5Controller=? -1, SignalTarget=LCFA_profile 1
EventTableEntry 8095: Group=, Trigger=pallet1.1 8096, Actions=[Pallet5.3 8097], Comment=, ActivationMode=2, Cyclic=false
EventTableTriggerIO 8096: IOValue=[1], IRC5Controller=? -1, Operator=0, SignalSource=LCFA_profile 1
EventTableActionIO 8097: IOValue=[0], IRC5Controller=? -1, SignalTarget=LCFA_profile 1
EventTableEntry 8098: Group=, Trigger=pallet1.1 8099, Actions=[Pallet5.4 8100], Comment=, ActivationMode=2, Cyclic=false
EventTableTriggerIO 8099: IOValue=[1], IRC5Controller=? -1, Operator=0, SignalSource=LCFA_profile 1
EventTableActionIO 8100: IOValue=[0], IRC5Controller=? -1, SignalTarget=LCFA_profile 1
EventTableEntry 8101: Group=, Trigger=pallet1.1 8102, Actions=[Pallet5.5 8103], Comment=, ActivationMode=2, Cyclic=false
EventTableTriggerIO 8102: IOValue=[1], IRC5Controller=? -1, Operator=0, SignalSource=LCFA_profile 1
EventTableActionIO 8103: IOValue=[0], IRC5Controller=? -1, SignalTarget=LCFA_profile 1
EventTableEntry 8104: Group=, Trigger=pallet1.1 8105, Actions=[Pallet5.6 8106], Comment=, ActivationMode=2, Cyclic=false
EventTableTriggerIO 8105: IOValue=[1], IRC5Controller=? -1, Operator=0, SignalSource=LCFA_profile 1
EventTableActionIO 8106: IOValue=[0], IRC5Controller=? -1, SignalTarget=LCFA_profile 1
EventTableEntry 8107: Group=, Trigger=pallet1.1 8108, Actions=[Pallet5.7 8109], Comment=, ActivationMode=2, Cyclic=false
EventTableTriggerIO 8108: IOValue=[1], IRC5Controller=? -1, Operator=0, SignalSource=LCFA_profile 1
EventTableActionIO 8109: IOValue=[0], IRC5Controller=? -1, SignalTarget=LCFA_profile 1
EventTableEntry 8110: Group=, Trigger=pallet1.1 8111, Actions=[Pallet5.8 8112], Comment=, ActivationMode=2, Cyclic=false
EventTableTriggerIO 8111: IOValue=[1], IRC5Controller=? -1, Operator=0, SignalSource=LCFA_profile 1
EventTableActionIO 8112: IOValue=[0], IRC5Controller=? -1, SignalTarget=LCFA_profile 1
EventTableTriggerLogic 8113: layoutX=251, layoutY=143, Operand1=AND 8115, Operand2=pallet3.1 8114, Operator=0, Delay=1000
EventTableTriggerIO 8114: IOValue=[-1], IRC5Controller=? -1, Operator=0, SignalSource=LCFA_profile 1
EventTableTriggerLogic 8115: layoutX=168, layoutY=75, Operand1=AND 8116, Operand2=AND 8120, Operator=0, Delay=1000
EventTableTriggerLogic 8116: layoutX=82, layoutY=32, Operand1=conv1_motor_s1 8117, Operand2=NOT 8118, Operator=0, Delay=1000
EventTableTriggerIO 8117: IOValue=[-1], IRC5Controller=? -1, Operator=0, SignalSource=ALab_CellC_v1.0_4 5362
EventTableTriggerLogic 8118: layoutX=22, layoutY=54, Operand1=conv1_motor_s2 8119, Operand2=? -1, Operator=2, Delay=1000
EventTableTriggerIO 8119: IOValue=[-1], IRC5Controller=? -1, Operator=0, SignalSource=ALab_CellC_v1.0_4 5362
EventTableTriggerLogic 8120: layoutX=102, layoutY=108, Operand1=NOT 8121, Operand2=NOT 8123, Operator=0, Delay=1000
EventTableTriggerLogic 8121: layoutX=21, layoutY=97, Operand1=conv2_motor_s1 8122, Operand2=? -1, Operator=2, Delay=1000
EventTableTriggerIO 8122: IOValue=[-1], IRC5Controller=? -1, Operator=0, SignalSource=ALab_CellC_v1.0_4 5362
EventTableTriggerLogic 8123: layoutX=27, layoutY=133, Operand1=conv2_motor_s2 8124, Operand2=? -1, Operator=2, Delay=1000
EventTableTriggerIO 8124: IOValue=[-1], IRC5Controller=? -1, Operator=0, SignalSource=ALab_CellC_v1.0_4 5362
EventTableTriggerIO 8125: IOValue=[-1], IRC5Controller=? -1, Operator=0, SignalSource=ALab_CellC_v1.0_4 5362
EventTableTriggerIO 8126: IOValue=[-1], IRC5Controller=? -1, Operator=0, SignalSource=LCFA_profile 1
EventTableTriggerIO 8127: IOValue=[-1], IRC5Controller=? -1, Operator=0, SignalSource=ALab_CellC_v1.0_4 5362
EventTableTriggerIO 8128: IOValue=[-1], IRC5Controller=? -1, Operator=0, SignalSource=ALab_CellC_v1.0_4 5362
EventTableTriggerIO 8133: IOValue=[-1], IRC5Controller=? -1, Operator=0, SignalSource=ALab_CellC_v1.0_4 5362
EventTableTriggerIO 8134: IOValue=[-1], IRC5Controller=? -1, Operator=0, SignalSource=ALab_CellC_v1.0_4 5362
EventTableTriggerLogic 8135: layoutX=8, layoutY=16, Operand1=conv2_buffer_upper_vertical_move 8136, Operand2=? -1, Operator=2, Delay=1000
EventTableTriggerIO 8136: IOValue=[-1], IRC5Controller=? -1, Operator=0, SignalSource=ALab_CellC_v1.0_4 5362
EventTableEntry 8137: Group=, Trigger=AND 8138, Actions=[PalletIO24 8142], Comment=, ActivationMode=2, Cyclic=false
EventTableTriggerLogic 8138: layoutX=99, layoutY=32, Operand1=Pallet2.1 8141, Operand2=NOT 8139, Operator=0, Delay=1000
EventTableTriggerLogic 8139: layoutX=37, layoutY=80, Operand1=conv1_buffer_horizontal_open 8140, Operand2=? -1, Operator=2, Delay=1000
EventTableTriggerIO 8140: IOValue=[-1], IRC5Controller=? -1, Operator=0, SignalSource=ALab_CellC_v1.0_4 5362
EventTableTriggerIO 8141: IOValue=[-1], IRC5Controller=? -1, Operator=0, SignalSource=LCFA_profile 1
EventTableActionIO 8142: IOValue=[-1], IRC5Controller=? -1, SignalTarget=LCFA_profile 1
EventTableEntry 8143: Group=, Trigger=AND 8144, Actions=[PalletIO25 8147], Comment=, ActivationMode=2, Cyclic=false
EventTableTriggerLogic 8144: layoutX=181, layoutY=52, Operand1=conv1_buffer_upper_go_down 8146, Operand2=Pallet2.2 8145, Operator=0, Delay=1000
EventTableTriggerIO 8145: IOValue=[-1], IRC5Controller=? -1, Operator=0, SignalSource=LCFA_profile 1
EventTableTriggerIO 8146: IOValue=[-1], IRC5Controller=? -1, Operator=0, SignalSource=ALab_CellC_v1.0_4 5362
EventTableActionIO 8147: IOValue=[-1], IRC5Controller=? -1, SignalTarget=LCFA_profile 1
EventTableEntry 8148: Group=, Trigger=AND 8149, Actions=[PalletIO26 8152], Comment=, ActivationMode=2, Cyclic=false
EventTableTriggerLogic 8149: layoutX=48, layoutY=51, Operand1=Pallet2.3 8150, Operand2=conv1_buffer_lower_go_up 8151, Operator=0, Delay=1000
EventTableTriggerIO 8150: IOValue=[-1], IRC5Controller=? -1, Operator=0, SignalSource=LCFA_profile 1
EventTableTriggerIO 8151: IOValue=[-1], IRC5Controller=? -1, Operator=0, SignalSource=ALab_CellC_v1.0_4 5362
EventTableActionIO 8152: IOValue=[-1], IRC5Controller=? -1, SignalTarget=LCFA_profile 1
EventTableEntry 8153: Group=, Trigger=AND 8154, Actions=[PalletIO23 8158], Comment=, ActivationMode=2, Cyclic=false
EventTableTriggerLogic 8154: layoutX=67, layoutY=33, Operand1=pallet2 8155, Operand2=NOT 8156, Operator=0, Delay=1000
EventTableTriggerIO 8155: IOValue=[-1], IRC5Controller=? -1, Operator=0, SignalSource=LCFA_profile 1
EventTableTriggerLogic 8156: layoutX=7, layoutY=52, Operand1=conv1_buffer_upper_go_down 8157, Operand2=? -1, Operator=2, Delay=1000
EventTableTriggerIO 8157: IOValue=[-1], IRC5Controller=? -1, Operator=0, SignalSource=ALab_CellC_v1.0_4 5362
EventTableActionIO 8158: IOValue=[-1], IRC5Controller=? -1, SignalTarget=LCFA_profile 1
EventTableEntry 8159: Group=, Trigger=AND 8160, Actions=[PalletIO27 8164], Comment=, ActivationMode=2, Cyclic=false
EventTableTriggerLogic 8160: layoutX=102, layoutY=29, Operand1=Pallet2.4 8161, Operand2=NOT 8162, Operator=0, Delay=1000
EventTableTriggerIO 8161: IOValue=[-1], IRC5Controller=? -1, Operator=0, SignalSource=LCFA_profile 1
EventTableTriggerLogic 8162: layoutX=16, layoutY=35, Operand1=conv1_buffer_lower_go_up 8163, Operand2=? -1, Operator=2, Delay=1000
EventTableTriggerIO 8163: IOValue=[-1], IRC5Controller=? -1, Operator=0, SignalSource=ALab_CellC_v1.0_4 5362
EventTableActionIO 8164: IOValue=[-1], IRC5Controller=? -1, SignalTarget=LCFA_profile 1
EventTableEntry 8165: Group=, Trigger=AND 8166, Actions=[PalletIO28 8170], Comment=, ActivationMode=2, Cyclic=false
EventTableTriggerLogic 8166: layoutX=102, layoutY=23, Operand1=Pallet2.5 8167, Operand2=NOT 8168, Operator=0, Delay=1000
EventTableTriggerIO 8167: IOValue=[-1], IRC5Controller=? -1, Operator=0, SignalSource=LCFA_profile 1
EventTableTriggerLogic 8168: layoutX=31, layoutY=54, Operand1=conv1_buffer_upper_go_down 8169, Operand2=? -1, Operator=2, Delay=1000
EventTableTriggerIO 8169: IOValue=[-1], IRC5Controller=? -1, Operator=0, SignalSource=ALab_CellC_v1.0_4 5362
EventTableActionIO 8170: IOValue=[-1], IRC5Controller=? -1, SignalTarget=LCFA_profile 1
EventTableEntry 8171: Group=, Trigger=PalletIO23 8172, Actions=[Pallet2.1 8173], Comment=, ActivationMode=2, Cyclic=false
EventTableTriggerIO 8172: IOValue=[1], IRC5Controller=? -1, Operator=0, SignalSource=LCFA_profile 1
EventTableActionIO 8173: IOValue=[1], IRC5Controller=? -1, SignalTarget=LCFA_profile 1
EventTableEntry 8174: Group=, Trigger=PalletIO24 8175, Actions=[Pallet2.2 8176], Comment=, ActivationMode=2, Cyclic=false
EventTableTriggerIO 8175: IOValue=[1], IRC5Controller=? -1, Operator=0, SignalSource=LCFA_profile 1
EventTableActionIO 8176: IOValue=[1], IRC5Controller=? -1, SignalTarget=LCFA_profile 1
EventTableEntry 8177: Group=, Trigger=PalletIO25 8178, Actions=[Pallet2.3 8179], Comment=, ActivationMode=2, Cyclic=false
EventTableTriggerIO 8178: IOValue=[1], IRC5Controller=? -1, Operator=0, SignalSource=LCFA_profile 1
EventTableActionIO 8179: IOValue=[1], IRC5Controller=? -1, SignalTarget=LCFA_profile 1
EventTableEntry 8180: Group=, Trigger=PalletIO26 8181, Actions=[Pallet2.4 8182], Comment=, ActivationMode=2, Cyclic=false
EventTableTriggerIO 8181: IOValue=[1], IRC5Controller=? -1, Operator=0, SignalSource=LCFA_profile 1
EventTableActionIO 8182: IOValue=[1], IRC5Controller=? -1, SignalTarget=LCFA_profile 1
EventTableEntry 8183: Group=, Trigger=PalletIO28 8184, Actions=[Pallet2.6 8185], Comment=, ActivationMode=2, Cyclic=false
EventTableTriggerIO 8184: IOValue=[1], IRC5Controller=? -1, Operator=0, SignalSource=LCFA_profile 1
EventTableActionIO 8185: IOValue=[1], IRC5Controller=? -1, SignalTarget=LCFA_profile 1
EventTableEntry 8186: Group=, Trigger=PalletIO27 8187, Actions=[Pallet2.5 8188], Comment=, ActivationMode=2, Cyclic=false
EventTableTriggerIO 8187: IOValue=[1], IRC5Controller=? -1, Operator=0, SignalSource=LCFA_profile 1
EventTableActionIO 8188: IOValue=[1], IRC5Controller=? -1, SignalTarget=LCFA_profile 1
EventTableEntry 8189: Group=, Trigger=Pallet2.1 8190, Actions=[pallet2 8191], Comment=, ActivationMode=2, Cyclic=false
EventTableTriggerIO 8190: IOValue=[1], IRC5Controller=? -1, Operator=0, SignalSource=LCFA_profile 1
EventTableActionIO 8191: IOValue=[0], IRC5Controller=? -1, SignalTarget=LCFA_profile 1
EventTableEntry 8192: Group=, Trigger=Pallet2.4 8193, Actions=[pickpallet4 8194], Comment=, ActivationMode=2, Cyclic=false
EventTableTriggerIO 8193: IOValue=[1], IRC5Controller=? -1, Operator=0, SignalSource=LCFA_profile 1
EventTableActionIO 8194: IOValue=[1], IRC5Controller=? -1, SignalTarget=LCFA_profile 1
EventTableEntry 8195: Group=, Trigger=pallet1.1 8196, Actions=[Pallet2.1 8197], Comment=, ActivationMode=2, Cyclic=false
EventTableTriggerIO 8196: IOValue=[1], IRC5Controller=? -1, Operator=0, SignalSource=LCFA_profile 1
EventTableActionIO 8197: IOValue=[0], IRC5Controller=? -1, SignalTarget=LCFA_profile 1
EventTableEntry 8198: Group=, Trigger=pallet1.1 8199, Actions=[Pallet2.2 8200], Comment=, ActivationMode=2, Cyclic=false
EventTableTriggerIO 8199: IOValue=[1], IRC5Controller=? -1, Operator=0, SignalSource=LCFA_profile 1
EventTableActionIO 8200: IOValue=[0], IRC5Controller=? -1, SignalTarget=LCFA_profile 1
EventTableEntry 8201: Group=, Trigger=pallet1.1 8202, Actions=[Pallet2.3 8203], Comment=, ActivationMode=2, Cyclic=false
EventTableTriggerIO 8202: IOValue=[1], IRC5Controller=? -1, Operator=0, SignalSource=LCFA_profile 1
EventTableActionIO 8203: IOValue=[0], IRC5Controller=? -1, SignalTarget=LCFA_profile 1
EventTableEntry 8204: Group=, Trigger=pallet1.1 8205, Actions=[Pallet2.4 8206], Comment=, ActivationMode=2, Cyclic=false
EventTableTriggerIO 8205: IOValue=[1], IRC5Controller=? -1, Operator=0, SignalSource=LCFA_profile 1
EventTableActionIO 8206: IOValue=[0], IRC5Controller=? -1, SignalTarget=LCFA_profile 1
EventTableEntry 8207: Group=, Trigger=pallet1.1 8208, Actions=[Pallet2.5 8209], Comment=, ActivationMode=2, Cyclic=false
EventTableTriggerIO 8208: IOValue=[1], IRC5Controller=? -1, Operator=0, SignalSource=LCFA_profile 1
EventTableActionIO 8209: IOValue=[0], IRC5Controller=? -1, SignalTarget=LCFA_profile 1
EventTableEntry 8210: Group=, Trigger=AND 8212, Actions=[PalletIO29 8211], Comment=, ActivationMode=2, Cyclic=false
EventTableActionIO 8211: IOValue=[-1], IRC5Controller=? -1, SignalTarget=LCFA_profile 1
EventTableTriggerLogic 8212: layoutX=49, layoutY=26, Operand1=Pallet2.6 8213, Operand2=conv1_buffer_horizontal_open 8214, Operator=0, Delay=1000
EventTableTriggerIO 8213: IOValue=[-1], IRC5Controller=? -1, Operator=0, SignalSource=LCFA_profile 1
EventTableTriggerIO 8214: IOValue=[-1], IRC5Controller=? -1, Operator=0, SignalSource=ALab_CellC_v1.0_4 5362
EventTableEntry 8215: Group=, Trigger=PalletIO29 8216, Actions=[pallet2 8217], Comment=, ActivationMode=2, Cyclic=false
EventTableTriggerIO 8216: IOValue=[1], IRC5Controller=? -1, Operator=0, SignalSource=LCFA_profile 1
EventTableActionIO 8217: IOValue=[1], IRC5Controller=? -1, SignalTarget=LCFA_profile 1
EventTableEntry 8218: Group=, Trigger=pallet2 8219, Actions=[conv1_pallet_buffer 8220], Comment=, ActivationMode=2, Cyclic=false
EventTableTriggerIO 8219: IOValue=[1], IRC5Controller=? -1, Operator=0, SignalSource=LCFA_profile 1
EventTableActionIO 8220: IOValue=[1], IRC5Controller=? -1, SignalTarget=ALab_CellC_v1.0_4 5362
EventTableEntry 8221: Group=, Trigger=pallet3 8222, Actions=[conv1_pallet_buffer 8223], Comment=, ActivationMode=2, Cyclic=false
EventTableTriggerIO 8222: IOValue=[1], IRC5Controller=? -1, Operator=0, SignalSource=LCFA_profile 1
EventTableActionIO 8223: IOValue=[0], IRC5Controller=? -1, SignalTarget=ALab_CellC_v1.0_4 5362
EventTableEntry 8224: Group=, Trigger=pallet6 8225, Actions=[conv2_pallet_buffer 8226], Comment=, ActivationMode=2, Cyclic=false
EventTableTriggerIO 8225: IOValue=[1], IRC5Controller=? -1, Operator=0, SignalSource=LCFA_profile 1
EventTableActionIO 8226: IOValue=[0], IRC5Controller=? -1, SignalTarget=ALab_CellC_v1.0_4 5362
EventTableEntry 8227: Group=, Trigger=pallet5 8228, Actions=[conv2_pallet_buffer 8229], Comment=, ActivationMode=2, Cyclic=false
EventTableTriggerIO 8228: IOValue=[1], IRC5Controller=? -1, Operator=0, SignalSource=LCFA_profile 1
EventTableActionIO 8229: IOValue=[1], IRC5Controller=? -1, SignalTarget=ALab_CellC_v1.0_4 5362
EventTableEntry 8230: Group=, Trigger=conv1_buffer_horizontal_open 8231, Actions=[conv1_pallet_lifter_in 8232], Comment=, ActivationMode=2, Cyclic=false
EventTableTriggerIO 8231: IOValue=[1], IRC5Controller=? -1, Operator=0, SignalSource=ALab_CellC_v1.0_4 5362
EventTableActionIO 8232: IOValue=[1], IRC5Controller=? -1, SignalTarget=ALab_CellC_v1.0_4 5362
EventTableEntry 8233: Group=, Trigger=conv1_buffer_horizontal_open 8234, Actions=[conv1_pallet_lifter_in 8235], Comment=, ActivationMode=2, Cyclic=false
EventTableTriggerIO 8234: IOValue=[0], IRC5Controller=? -1, Operator=0, SignalSource=ALab_CellC_v1.0_4 5362
EventTableActionIO 8235: IOValue=[0], IRC5Controller=? -1, SignalTarget=ALab_CellC_v1.0_4 5362
EventTableEntry 8236: Group=, Trigger=conv1_buffer_horizontal_open 8237, Actions=[conv1_pallet_lifter_out 8238], Comment=, ActivationMode=2, Cyclic=false
EventTableTriggerIO 8237: IOValue=[1], IRC5Controller=? -1, Operator=0, SignalSource=ALab_CellC_v1.0_4 5362
EventTableActionIO 8238: IOValue=[0], IRC5Controller=? -1, SignalTarget=ALab_CellC_v1.0_4 5362
